LIN {X 0,Y 627.245,Z 767.06,A -85,B 0,C 180,E1 6657.903,E2 6657.903} C_VEL
LIN {X 0,Y 626.761,Z 767.06,A -85,B 0,C 180,E1 6666.234,E2 6666.234} C_VEL
LIN {X 0,Y 626.409,Z 767.06,A -85,B 0,C 180,E1 6674.712,E2 6674.712} C_VEL
LIN {X 0,Y 626.287,Z 767.06,A -85,B 0,C 180,E1 6682.031,E2 6682.031} C_VEL
LIN {X 0,Y 626.18,Z 767.06,A -85,B 0,C 180,E1 6690.73,E2 6690.73} C_VEL
LIN {X 0,Y 626.045,Z 767.06,A -85,B 0,C 180,E1 6698.138,E2 6698.138} C_VEL
LIN {X 0,Y 626.097,Z 767.06,A -85,B 0,C 180,E1 6703.652,E2 6703.652} C_VEL
LIN {X 0,Y 628.32,Z 775.547,A -85,B 0,C 180,E1 6704.191,E2 6704.191} C_VEL
LIN {X 0,Y 630.234,Z 788.438,A -85,B 0,C 180,E1 6704.573,E2 6704.573} C_VEL
LIN {X 0,Y 651.421,Z 829.278,A -85,B 0,C 180,E1 6707.069,E2 6707.069} C_VEL
LIN {X 0,Y 646.587,Z 907.539,A -85,B 0,C 180,E1 6708.986,E2 6708.986} C_VEL
LIN {X 0,Y 639.747,Z 982.775,A -85,B 0,C 180,E1 6712.403,E2 6712.403} C_VEL
LIN {X 0,Y 632.395,Z 1050.27,A -85,B 0,C 180,E1 6717.121,E2 6717.121} C_VEL
LIN {X 0,Y 626.259,Z 1107.378,A -85,B 0,C 180,E1 6722.867,E2 6722.867} C_VEL
LIN {X 0,Y 622.003,Z 1154.489,A -85,B 0,C 180,E1 6729.657,E2 6729.657} C_VEL
LIN {X 0,Y 619.694,Z 1186.305,A -85,B 0,C 180,E1 6736.585,E2 6736.585} C_VEL
LIN {X 0,Y 619.248,Z 1202.946,A -85,B 0,C 180,E1 6742.653,E2 6742.653} C_VEL
LIN {X 0,Y 619.266,Z 1209.424,A -85,B 0,C 180,E1 6747.928,E2 6747.928} C_VEL
LIN {X 0,Y 619.05,Z 1206.761,A -85,B 0,C 180,E1 6754.956,E2 6754.956} C_VEL
LIN {X 0,Y 619.262,Z 1193.655,A -85,B 0,C 180,E1 6761.174,E2 6761.174} C_VEL
LIN {X 0,Y 620.519,Z 1169.572,A -85,B 0,C 180,E1 6767.441,E2 6767.441} C_VEL
LIN {X 0,Y 623.271,Z 1133.468,A -85,B 0,C 180,E1 6773.72,E2 6773.72} C_VEL
LIN {X 0,Y 628.625,Z 1081.833,A -85,B 0,C 180,E1 6779.974,E2 6779.974} C_VEL
LIN {X 0,Y 635.923,Z 1018.771,A -85,B 0,C 180,E1 6785.31,E2 6785.31} C_VEL
LIN {X 0,Y 643.31,Z 949.028,A -85,B 0,C 180,E1 6789.325,E2 6789.325} C_VEL
LIN {X 0,Y 649.136,Z 874.323,A -85,B 0,C 180,E1 6792.011,E2 6792.011} C_VEL
LIN {X 0,Y 650.044,Z 823.777,A -85,B 0,C 180,E1 6793.141,E2 6793.141} C_VEL
LIN {X 0,Y 618.157,Z 767.06,A -85,B 0,C 180,E1 6797.036,E2 6797.036} C_VEL
LIN {X 0,Y 618.384,Z 767.06,A -85,B 0,C 180,E1 6806.522,E2 6806.522} C_VEL
LIN {X 0,Y 618.649,Z 767.06,A -85,B 0,C 180,E1 6814.61,E2 6814.61} C_VEL
LIN {X 0,Y 618.58,Z 767.06,A -85,B 0,C 180,E1 6823.639,E2 6823.639} C_VEL
LIN {X 0,Y 618.828,Z 767.06,A -85,B 0,C 180,E1 6832.27,E2 6832.27} C_VEL
LIN {X 0,Y 618.766,Z 767.06,A -85,B 0,C 180,E1 6840.721,E2 6840.721} C_VEL
LIN {X 0,Y 618.86,Z 767.06,A -85,B 0,C 180,E1 6847.767,E2 6847.767} C_VEL
LIN {X 0,Y 618.363,Z 767.06,A -85,B 0,C 180,E1 6856.406,E2 6856.406} C_VEL
LIN {X 0,Y 618.222,Z 767.06,A -85,B 0,C 180,E1 6865.45,E2 6865.45} C_VEL
LIN {X 0,Y 618.091,Z 767.06,A -85,B 0,C 180,E1 6873.541,E2 6873.541} C_VEL
LIN {X 0,Y 618.177,Z 767.06,A -85,B 0,C 180,E1 6882.465,E2 6882.465} C_VEL
LIN {X 0,Y 618.232,Z 768.464,A -85,B 0,C 180,E1 6890.217,E2 6890.217} C_VEL
LIN {X 0,Y 651.124,Z 828.1,A -85,B 0,C 180,E1 6894.171,E2 6894.171} C_VEL
LIN {X 0,Y 646.571,Z 901.597,A -85,B 0,C 180,E1 6896.097,E2 6896.097} C_VEL
LIN {X 0,Y 639.646,Z 974.672,A -85,B 0,C 180,E1 6899.467,E2 6899.467} C_VEL
LIN {X 0,Y 632.064,Z 1042.701,A -85,B 0,C 180,E1 6904.278,E2 6904.278} C_VEL
LIN {X 0,Y 625.576,Z 1101.407,A -85,B 0,C 180,E1 6910.298,E2 6910.298} C_VEL
LIN {X 0,Y 621.333,Z 1147.196,A -85,B 0,C 180,E1 6917.086,E2 6917.086} C_VEL
LIN {X 0,Y 619.437,Z 1176.669,A -85,B 0,C 180,E1 6923.637,E2 6923.637} C_VEL
LIN {X 0,Y 618.869,Z 1193.621,A -85,B 0,C 180,E1 6929.965,E2 6929.965} C_VEL
LIN {X 0,Y 618.768,Z 1199.851,A -85,B 0,C 180,E1 6936.3,E2 6936.3} C_VEL
LIN {X 0,Y 618.868,Z 1195.665,A -85,B 0,C 180,E1 6942.712,E2 6942.712} C_VEL
LIN {X 0,Y 619.249,Z 1179.816,A -85,B 0,C 180,E1 6949.363,E2 6949.363} C_VEL
LIN {X 0,Y 620.829,Z 1153.329,A -85,B 0,C 180,E1 6955.671,E2 6955.671} C_VEL
LIN {X 0,Y 624.482,Z 1111.503,A -85,B 0,C 180,E1 6962.324,E2 6962.324} C_VEL
LIN {X 0,Y 630.592,Z 1055.076,A -85,B 0,C 180,E1 6968.544,E2 6968.544} C_VEL
LIN {X 0,Y 638.132,Z 989.06,A -85,B 0,C 180,E1 6973.576,E2 6973.576} C_VEL
LIN {X 0,Y 645.271,Z 917.737,A -85,B 0,C 180,E1 6977.198,E2 6977.198} C_VEL
LIN {X 0,Y 650.203,Z 848.201,A -85,B 0,C 180,E1 6979.337,E2 6979.337} C_VEL
LIN {X 0,Y 649.666,Z 822.506,A -85,B 0,C 180,E1 6979.978,E2 6979.978} C_VEL
LIN {X 0,Y 618.29,Z 767.06,A -85,B 0,C 180,E1 6983.94,E2 6983.94} C_VEL
LIN {X 0,Y 618.29,Z 767.06,A -85,B 0,C 180,E1 6992.986,E2 6992.986} C_VEL
LIN {X 0,Y 618.359,Z 767.06,A -85,B 0,C 180,E1 7000.747,E2 7000.747} C_VEL
LIN {X 0,Y 619.19,Z 767.06,A -85,B 0,C 180,E1 7009.393,E2 7009.393} C_VEL
LIN {X 0,Y 619.243,Z 767.06,A -85,B 0,C 180,E1 7017.876,E2 7017.876} C_VEL
LIN {X 0,Y 618.542,Z 767.06,A -85,B 0,C 180,E1 7026.854,E2 7026.854} C_VEL
LIN {X 0,Y 618.36,Z 767.06,A -85,B 0,C 180,E1 7034.908,E2 7034.908} C_VEL
LIN {X 0,Y 618.08,Z 767.06,A -85,B 0,C 180,E1 7043.081,E2 7043.081} C_VEL
LIN {X 0,Y 618.03,Z 767.06,A -85,B 0,C 180,E1 7051.829,E2 7051.829} C_VEL
LIN {X 0,Y 617.761,Z 767.06,A -85,B 0,C 180,E1 7060.572,E2 7060.572} C_VEL
LIN {X 0,Y 618.103,Z 768.608,A -85,B 0,C 180,E1 7063.099,E2 7063.099} C_VEL
LIN {X 0,Y 630.234,Z 788.438,A -85,B 0,C 180,E1 7064.573,E2 7064.573} C_VEL
LIN {X 0,Y 635.159,Z 810.265,A -85,B 0,C 180,E1 7065.359,E2 7065.359} C_VEL
LIN {X 0,Y 645.533,Z 832.217,A -85,B 0,C 180,E1 7066.634,E2 7066.634} C_VEL
LIN {X 0,Y 640.352,Z 909.412,A -85,B 0,C 180,E1 7068.575,E2 7068.575} C_VEL
LIN {X 0,Y 633.189,Z 982.863,A -85,B 0,C 180,E1 7071.95,E2 7071.95} C_VEL
LIN {X 0,Y 625.431,Z 1049.905,A -85,B 0,C 180,E1 7076.674,E2 7076.674} C_VEL
LIN {X 0,Y 618.742,Z 1107.804,A -85,B 0,C 180,E1 7082.563,E2 7082.563} C_VEL
LIN {X 0,Y 614.293,Z 1154.485,A -85,B 0,C 180,E1 7089.389,E2 7089.389} C_VEL
LIN {X 0,Y 611.622,Z 1187.618,A -85,B 0,C 180,E1 7096.77,E2 7096.77} C_VEL
LIN {X 0,Y 610.939,Z 1204.79,A -85,B 0,C 180,E1 7103.619,E2 7103.619} C_VEL
LIN {X 0,Y 610.73,Z 1209.846,A -85,B 0,C 180,E1 7109.323,E2 7109.323} C_VEL
LIN {X 0,Y 610.928,Z 1205.826,A -85,B 0,C 180,E1 7115.737,E2 7115.737} C_VEL
LIN {X 0,Y 611.291,Z 1190.908,A -85,B 0,C 180,E1 7122.215,E2 7122.215} C_VEL
LIN {X 0,Y 612.788,Z 1165.943,A -85,B 0,C 180,E1 7128.439,E2 7128.439} C_VEL
LIN {X 0,Y 616.388,Z 1126.344,A -85,B 0,C 180,E1 7135.04,E2 7135.04} C_VEL
LIN {X 0,Y 622.443,Z 1072.303,A -85,B 0,C 180,E1 7141.31,E2 7141.31} C_VEL
LIN {X 0,Y 630.415,Z 1007.933,A -85,B 0,C 180,E1 7146.495,E2 7146.495} C_VEL
LIN {X 0,Y 638.116,Z 938.064,A -85,B 0,C 180,E1 7150.277,E2 7150.277} C_VEL
LIN {X 0,Y 643.685,Z 867.024,A -85,B 0,C 180,E1 7152.661,E2 7152.661} C_VEL
LIN {X 0,Y 644.21,Z 827.262,A -85,B 0,C 180,E1 7153.566,E2 7153.566} C_VEL
LIN {X 0,Y 610.074,Z 767.06,A -85,B 0,C 180,E1 7157.871,E2 7157.871} C_VEL
LIN {X 0,Y 610.378,Z 767.06,A -85,B 0,C 180,E1 7166.445,E2 7166.445} C_VEL
LIN {X 0,Y 610.572,Z 767.06,A -85,B 0,C 180,E1 7175.181,E2 7175.181} C_VEL
LIN {X 0,Y 610.494,Z 767.06,A -85,B 0,C 180,E1 7184.896,E2 7184.896} C_VEL
LIN {X 0,Y 610.475,Z 767.06,A -85,B 0,C 180,E1 7193.599,E2 7193.599} C_VEL
LIN {X 0,Y 610.759,Z 767.06,A -85,B 0,C 180,E1 7200.73,E2 7200.73} C_VEL
LIN {X 0,Y 610.807,Z 767.06,A -85,B 0,C 180,E1 7207.87,E2 7207.87} C_VEL
LIN {X 0,Y 610.277,Z 767.06,A -85,B 0,C 180,E1 7216.704,E2 7216.704} C_VEL
LIN {X 0,Y 610.235,Z 767.06,A -85,B 0,C 180,E1 7224.751,E2 7224.751} C_VEL
LIN {X 0,Y 610.105,Z 767.06,A -85,B 0,C 180,E1 7233.517,E2 7233.517} C_VEL
LIN {X 0,Y 610.171,Z 767.06,A -85,B 0,C 180,E1 7242.763,E2 7242.763} C_VEL
LIN {X 0,Y 610.117,Z 768.406,A -85,B 0,C 180,E1 7249.401,E2 7249.401} C_VEL
LIN {X 0,Y 645.164,Z 829.949,A -85,B 0,C 180,E1 7253.722,E2 7253.722} C_VEL
LIN {X 0,Y 640.323,Z 902.679,A -85,B 0,C 180,E1 7255.661,E2 7255.661} C_VEL
LIN {X 0,Y 632.989,Z 975.5,A -85,B 0,C 180,E1 7259.06,E2 7259.06} C_VEL
LIN {X 0,Y 625.052,Z 1042.571,A -85,B 0,C 180,E1 7263.853,E2 7263.853} C_VEL
LIN {X 0,Y 618.218,Z 1100.711,A -85,B 0,C 180,E1 7269.867,E2 7269.867} C_VEL
LIN {X 0,Y 613.633,Z 1146.761,A -85,B 0,C 180,E1 7276.743,E2 7276.743} C_VEL
LIN {X 0,Y 611.514,Z 1176.997,A -85,B 0,C 180,E1 7283.554,E2 7283.554} C_VEL
LIN {X 0,Y 610.885,Z 1193.782,A -85,B 0,C 180,E1 7289.965,E2 7289.965} C_VEL
LIN {X 0,Y 610.775,Z 1199.873,A -85,B 0,C 180,E1 7296.383,E2 7296.383} C_VEL
LIN {X 0,Y 610.899,Z 1195.518,A -85,B 0,C 180,E1 7302.88,E2 7302.88} C_VEL
LIN {X 0,Y 611.328,Z 1179.774,A -85,B 0,C 180,E1 7309.539,E2 7309.539} C_VEL
LIN {X 0,Y 613.078,Z 1152.806,A -85,B 0,C 180,E1 7316.019,E2 7316.019} C_VEL
LIN {X 0,Y 617.224,Z 1109.621,A -85,B 0,C 180,E1 7322.904,E2 7322.904} C_VEL
LIN {X 0,Y 623.652,Z 1053.919,A -85,B 0,C 180,E1 7329.053,E2 7329.053} C_VEL
LIN {X 0,Y 631.741,Z 986.989,A -85,B 0,C 180,E1 7334.155,E2 7334.155} C_VEL
LIN {X 0,Y 639.21,Z 915.736,A -85,B 0,C 180,E1 7337.752,E2 7337.752} C_VEL
LIN {X 0,Y 644.327,Z 847.615,A -85,B 0,C 180,E1 7339.831,E2 7339.831} C_VEL
LIN {X 0,Y 643.853,Z 826.122,A -85,B 0,C 180,E1 7340.385,E2 7340.385} C_VEL
LIN {X 0,Y 610.198,Z 767.06,A -85,B 0,C 180,E1 7344.645,E2 7344.645} C_VEL
LIN {X 0,Y 610.258,Z 767.06,A -85,B 0,C 180,E1 7352.601,E2 7352.601} C_VEL
LIN {X 0,Y 610.343,Z 767.06,A -85,B 0,C 180,E1 7360.375,E2 7360.375} C_VEL
LIN {X 0,Y 611.184,Z 767.06,A -85,B 0,C 180,E1 7369.253,E2 7369.253} C_VEL
LIN {X 0,Y 611.254,Z 767.06,A -85,B 0,C 180,E1 7377.848,E2 7377.848} C_VEL
LIN {X 0,Y 610.687,Z 767.06,A -85,B 0,C 180,E1 7386.399,E2 7386.399} C_VEL
LIN {X 0,Y 610.305,Z 767.06,A -85,B 0,C 180,E1 7395.109,E2 7395.109} C_VEL
LIN {X 0,Y 610.146,Z 767.06,A -85,B 0,C 180,E1 7402.646,E2 7402.646} C_VEL
LIN {X 0,Y 610.077,Z 767.06,A -85,B 0,C 180,E1 7410.973,E2 7410.973} C_VEL
LIN {X 0,Y 609.847,Z 767.06,A -85,B 0,C 180,E1 7419.343,E2 7419.343} C_VEL
LIN {X 0,Y 610.08,Z 768.922,A -85,B 0,C 180,E1 7422.298,E2 7422.298} C_VEL
LIN {X 0,Y 635.159,Z 810.265,A -85,B 0,C 180,E1 7425.359,E2 7425.359} C_VEL
LIN {X 0,Y 639.562,Z 835.031,A -85,B 0,C 180,E1 7426.178,E2 7426.178} C_VEL
LIN {X 0,Y 639.2,Z 843.944,A -85,B 0,C 180,E1 7426.355,E2 7426.355} C_VEL
LIN {X 0,Y 633.542,Z 919,A -85,B 0,C 180,E1 7428.451,E2 7428.451} C_VEL
LIN {X 0,Y 625.551,Z 992.775,A -85,B 0,C 180,E1 7432.078,E2 7432.078} C_VEL
LIN {X 0,Y 617.373,Z 1058.589,A -85,B 0,C 180,E1 7437.016,E2 7437.016} C_VEL
LIN {X 0,Y 610.525,Z 1114.591,A -85,B 0,C 180,E1 7443.061,E2 7443.061} C_VEL
LIN {X 0,Y 605.801,Z 1159.36,A -85,B 0,C 180,E1 7450.023,E2 7450.023} C_VEL
LIN {X 0,Y 603.549,Z 1188.827,A -85,B 0,C 180,E1 7456.96,E2 7456.96} C_VEL
LIN {X 0,Y 602.979,Z 1204.787,A -85,B 0,C 180,E1 7463.534,E2 7463.534} C_VEL
LIN {X 0,Y 602.732,Z 1209.846,A -85,B 0,C 180,E1 7469.314,E2 7469.314} C_VEL
LIN {X 0,Y 602.939,Z 1205.826,A -85,B 0,C 180,E1 7475.813,E2 7475.813} C_VEL
LIN {X 0,Y 603.328,Z 1190.905,A -85,B 0,C 180,E1 7482.379,E2 7482.379} C_VEL
LIN {X 0,Y 604.93,Z 1165.944,A -85,B 0,C 180,E1 7488.688,E2 7488.688} C_VEL
LIN {X 0,Y 608.833,Z 1125.749,A -85,B 0,C 180,E1 7495.46,E2 7495.46} C_VEL
LIN {X 0,Y 615.417,Z 1071.635,A -85,B 0,C 180,E1 7501.781,E2 7501.781} C_VEL
LIN {X 0,Y 623.853,Z 1007.033,A -85,B 0,C 180,E1 7507.013,E2 7507.013} C_VEL
LIN {X 0,Y 631.918,Z 937.652,A -85,B 0,C 180,E1 7510.776,E2 7510.776} C_VEL
LIN {X 0,Y 637.734,Z 867.851,A -85,B 0,C 180,E1 7513.131,E2 7513.131} C_VEL
LIN {X 0,Y 638.364,Z 830.573,A -85,B 0,C 180,E1 7514.006,E2 7514.006} C_VEL
LIN {X 0,Y 602.051,Z 767.06,A -85,B 0,C 180,E1 7518.785,E2 7518.785} C_VEL
LIN {X 0,Y 602.457,Z 767.06,A -85,B 0,C 180,E1 7527.598,E2 7527.598} C_VEL
LIN {X 0,Y 602.587,Z 767.06,A -85,B 0,C 180,E1 7535.478,E2 7535.478} C_VEL
LIN {X 0,Y 602.487,Z 767.06,A -85,B 0,C 180,E1 7544.69,E2 7544.69} C_VEL
LIN {X 0,Y 602.485,Z 767.06,A -85,B 0,C 180,E1 7553.513,E2 7553.513} C_VEL
LIN {X 0,Y 602.751,Z 767.06,A -85,B 0,C 180,E1 7560.74,E2 7560.74} C_VEL
LIN {X 0,Y 602.77,Z 767.06,A -85,B 0,C 180,E1 7567.975,E2 7567.975} C_VEL
LIN {X 0,Y 602.259,Z 767.06,A -85,B 0,C 180,E1 7576.857,E2 7576.857} C_VEL
LIN {X 0,Y 602.251,Z 767.06,A -85,B 0,C 180,E1 7584.578,E2 7584.578} C_VEL
LIN {X 0,Y 602.113,Z 767.06,A -85,B 0,C 180,E1 7592.82,E2 7592.82} C_VEL
LIN {X 0,Y 602.098,Z 767.06,A -85,B 0,C 180,E1 7601.926,E2 7601.926} C_VEL
LIN {X 0,Y 602.207,Z 768.812,A -85,B 0,C 180,E1 7608.58,E2 7608.58} C_VEL
LIN {X 0,Y 639.091,Z 832.378,A -85,B 0,C 180,E1 7613.264,E2 7613.264} C_VEL
LIN {X 0,Y 633.97,Z 905.735,A -85,B 0,C 180,E1 7615.294,E2 7615.294} C_VEL
LIN {X 0,Y 626.169,Z 978.142,A -85,B 0,C 180,E1 7618.756,E2 7618.756} C_VEL
LIN {X 0,Y 617.745,Z 1044.932,A -85,B 0,C 180,E1 7623.637,E2 7623.637} C_VEL
LIN {X 0,Y 610.474,Z 1102.98,A -85,B 0,C 180,E1 7629.79,E2 7629.79} C_VEL
LIN {X 0,Y 605.819,Z 1147.273,A -85,B 0,C 180,E1 7636.568,E2 7636.568} C_VEL
LIN {X 0,Y 603.594,Z 1177.326,A -85,B 0,C 180,E1 7643.469,E2 7643.469} C_VEL
LIN {X 0,Y 602.884,Z 1193.93,A -85,B 0,C 180,E1 7649.964,E2 7649.964} C_VEL
LIN {X 0,Y 602.78,Z 1199.894,A -85,B 0,C 180,E1 7656.468,E2 7656.468} C_VEL
LIN {X 0,Y 602.918,Z 1195.37,A -85,B 0,C 180,E1 7663.054,E2 7663.054} C_VEL
LIN {X 0,Y 603.442,Z 1179.466,A -85,B 0,C 180,E1 7669.805,E2 7669.805} C_VEL
LIN {X 0,Y 605.789,Z 1149.32,A -85,B 0,C 180,E1 7676.949,E2 7676.949} C_VEL
LIN {X 0,Y 610.52,Z 1104.186,A -85,B 0,C 180,E1 7683.956,E2 7683.956} C_VEL
LIN {X 0,Y 617.47,Z 1047.599,A -85,B 0,C 180,E1 7690.034,E2 7690.034} C_VEL
LIN {X 0,Y 625.867,Z 980.636,A -85,B 0,C 180,E1 7695.003,E2 7695.003} C_VEL
LIN {X 0,Y 633.785,Z 907.439,A -85,B 0,C 180,E1 7698.553,E2 7698.553} C_VEL
LIN {X 0,Y 639.125,Z 835.51,A -85,B 0,C 180,E1 7700.571,E2 7700.571} C_VEL
LIN {X 0,Y 612.906,Z 785.364,A -85,B 0,C 180,E1 7703.938,E2 7703.938} C_VEL
LIN {X 0,Y 602.132,Z 767.06,A -85,B 0,C 180,E1 7705.447,E2 7705.447} C_VEL
LIN {X 0,Y 602.207,Z 767.06,A -85,B 0,C 180,E1 7713.823,E2 7713.823} C_VEL
LIN {X 0,Y 602.301,Z 767.06,A -85,B 0,C 180,E1 7721.63,E2 7721.63} C_VEL
LIN {X 0,Y 603.206,Z 767.06,A -85,B 0,C 180,E1 7729.109,E2 7729.109} C_VEL
LIN {X 0,Y 603.25,Z 767.06,A -85,B 0,C 180,E1 7737.819,E2 7737.819} C_VEL
LIN {X 0,Y 602.65,Z 767.06,A -85,B 0,C 180,E1 7746.485,E2 7746.485} C_VEL
LIN {X 0,Y 602.256,Z 767.06,A -85,B 0,C 180,E1 7755.316,E2 7755.316} C_VEL
LIN {X 0,Y 602.056,Z 767.06,A -85,B 0,C 180,E1 7763.186,E2 7763.186} C_VEL
LIN {X 0,Y 602.073,Z 767.06,A -85,B 0,C 180,E1 7771.076,E2 7771.076} C_VEL
LIN {X 0,Y 601.779,Z 767.06,A -85,B 0,C 180,E1 7779.976,E2 7779.976} C_VEL
LIN {X 0,Y 601.935,Z 768.669,A -85,B 0,C 180,E1 7781.426,E2 7781.426} C_VEL
LIN {X 0,Y 639.583,Z 833.093,A -85,B 0,C 180,E1 7786.145,E2 7786.145} C_VEL
LIN {X 0,Y 639.2,Z 843.944,A -85,B 0,C 180,E1 7786.355,E2 7786.355} C_VEL
LIN {X 0,Y 631.176,Z 878.377,A -85,B 0,C 180,E1 7786.642,E2 7786.642} C_VEL
LIN {X 0,Y 624.414,Z 949.498,A -85,B 0,C 180,E1 7789.265,E2 7789.265} C_VEL
LIN {X 0,Y 615.761,Z 1018.278,A -85,B 0,C 180,E1 7793.312,E2 7793.312} C_VEL
LIN {X 0,Y 606.941,Z 1082.187,A -85,B 0,C 180,E1 7798.877,E2 7798.877} C_VEL
LIN {X 0,Y 600.372,Z 1133.976,A -85,B 0,C 180,E1 7805.394,E2 7805.394} C_VEL
LIN {X 0,Y 596.774,Z 1170.294,A -85,B 0,C 180,E1 7812,E2 7812} C_VEL
LIN {X 0,Y 595.208,Z 1193.25,A -85,B 0,C 180,E1 7818.224,E2 7818.224} C_VEL
LIN {X 0,Y 594.961,Z 1206.836,A -85,B 0,C 180,E1 7824.915,E2 7824.915} C_VEL
LIN {X 0,Y 594.613,Z 1209.829,A -85,B 0,C 180,E1 7830.767,E2 7830.767} C_VEL
LIN {X 0,Y 594.994,Z 1204.665,A -85,B 0,C 180,E1 7836.626,E2 7836.626} C_VEL
LIN {X 0,Y 595.769,Z 1187.377,A -85,B 0,C 180,E1 7843.662,E2 7843.662} C_VEL
LIN {X 0,Y 598.604,Z 1155.322,A -85,B 0,C 180,E1 7851.019,E2 7851.019} C_VEL
LIN {X 0,Y 603.669,Z 1109.45,A -85,B 0,C 180,E1 7857.973,E2 7857.973} C_VEL
LIN {X 0,Y 611.225,Z 1052.148,A -85,B 0,C 180,E1 7863.996,E2 7863.996} C_VEL
LIN {X 0,Y 620.033,Z 985.616,A -85,B 0,C 180,E1 7868.826,E2 7868.826} C_VEL
LIN {X 0,Y 628.218,Z 911.551,A -85,B 0,C 180,E1 7872.319,E2 7872.319} C_VEL
LIN {X 0,Y 632.404,Z 833.705,A -85,B 0,C 180,E1 7874.47,E2 7874.47} C_VEL
LIN {X 0,Y 596.309,Z 772.647,A -85,B 0,C 180,E1 7879.091,E2 7879.091} C_VEL
LIN {X 0,Y 594.044,Z 767.06,A -85,B 0,C 180,E1 7879.633,E2 7879.633} C_VEL
LIN {X 0,Y 594.49,Z 767.06,A -85,B 0,C 180,E1 7888.829,E2 7888.829} C_VEL
LIN {X 0,Y 594.409,Z 767.06,A -85,B 0,C 180,E1 7896.72,E2 7896.72} C_VEL
LIN {X 0,Y 594.331,Z 767.06,A -85,B 0,C 180,E1 7905.987,E2 7905.987} C_VEL
LIN {X 0,Y 594.496,Z 767.06,A -85,B 0,C 180,E1 7913.426,E2 7913.426} C_VEL
LIN {X 0,Y 594.751,Z 767.06,A -85,B 0,C 180,E1 7920.75,E2 7920.75} C_VEL
LIN {X 0,Y 594.722,Z 767.06,A -85,B 0,C 180,E1 7928.084,E2 7928.084} C_VEL
LIN {X 0,Y 594.233,Z 767.06,A -85,B 0,C 180,E1 7937.092,E2 7937.092} C_VEL
LIN {X 0,Y 594.206,Z 767.06,A -85,B 0,C 180,E1 7944.933,E2 7944.933} C_VEL
LIN {X 0,Y 594.014,Z 767.06,A -85,B 0,C 180,E1 7953.822,E2 7953.822} C_VEL
LIN {X 0,Y 594.061,Z 767.06,A -85,B 0,C 180,E1 7962.611,E2 7962.611} C_VEL
LIN {X 0,Y 594.184,Z 768.882,A -85,B 0,C 180,E1 7967.721,E2 7967.721} C_VEL
LIN {X 0,Y 632.996,Z 835.271,A -85,B 0,C 180,E1 7972.803,E2 7972.803} C_VEL
LIN {X 0,Y 627.613,Z 908.776,A -85,B 0,C 180,E1 7974.917,E2 7974.917} C_VEL
LIN {X 0,Y 619.346,Z 981.073,A -85,B 0,C 180,E1 7978.465,E2 7978.465} C_VEL
LIN {X 0,Y 610.427,Z 1047.351,A -85,B 0,C 180,E1 7983.42,E2 7983.42} C_VEL
LIN {X 0,Y 602.938,Z 1103.755,A -85,B 0,C 180,E1 7989.526,E2 7989.526} C_VEL
LIN {X 0,Y 598.024,Z 1147.784,A -85,B 0,C 180,E1 7996.39,E2 7996.39} C_VEL
LIN {X 0,Y 595.649,Z 1177.655,A -85,B 0,C 180,E1 8003.382,E2 8003.382} C_VEL
LIN {X 0,Y 594.889,Z 1194.078,A -85,B 0,C 180,E1 8009.964,E2 8009.964} C_VEL
LIN {X 0,Y 594.772,Z 1199.916,A -85,B 0,C 180,E1 8016.556,E2 8016.556} C_VEL
LIN {X 0,Y 594.972,Z 1195.22,A -85,B 0,C 180,E1 8023.231,E2 8023.231} C_VEL
LIN {X 0,Y 595.828,Z 1177.885,A -85,B 0,C 180,E1 8030.458,E2 8030.458} C_VEL
LIN {X 0,Y 598.642,Z 1145.555,A -85,B 0,C 180,E1 8037.922,E2 8037.922} C_VEL
LIN {X 0,Y 603.781,Z 1098.812,A -85,B 0,C 180,E1 8044.996,E2 8044.996} C_VEL
LIN {X 0,Y 611.28,Z 1042.076,A -85,B 0,C 180,E1 8050.95,E2 8050.95} C_VEL
LIN {X 0,Y 620.132,Z 974.657,A -85,B 0,C 180,E1 8055.839,E2 8055.839} C_VEL
LIN {X 0,Y 628.372,Z 899.804,A -85,B 0,C 180,E1 8059.344,E2 8059.344} C_VEL
LIN {X 0,Y 632.022,Z 833.034,A -85,B 0,C 180,E1 8061.246,E2 8061.246} C_VEL
LIN {X 0,Y 595.921,Z 772.134,A -85,B 0,C 180,E1 8065.99,E2 8065.99} C_VEL
LIN {X 0,Y 594.118,Z 767.06,A -85,B 0,C 180,E1 8066.387,E2 8066.387} C_VEL
LIN {X 0,Y 594.254,Z 767.06,A -85,B 0,C 180,E1 8075.069,E2 8075.069} C_VEL
LIN {X 0,Y 594.762,Z 767.06,A -85,B 0,C 180,E1 8084.446,E2 8084.446} C_VEL
LIN {X 0,Y 594.508,Z 767.06,A -85,B 0,C 180,E1 8091.913,E2 8091.913} C_VEL
LIN {X 0,Y 594.626,Z 767.06,A -85,B 0,C 180,E1 8099.25,E2 8099.25} C_VEL
LIN {X 0,Y 594.614,Z 767.06,A -85,B 0,C 180,E1 8106.573,E2 8106.573} C_VEL
LIN {X 0,Y 594.219,Z 767.06,A -85,B 0,C 180,E1 8115.528,E2 8115.528} C_VEL
LIN {X 0,Y 594.036,Z 767.06,A -85,B 0,C 180,E1 8123.296,E2 8123.296} C_VEL
LIN {X 0,Y 594.015,Z 767.06,A -85,B 0,C 180,E1 8131.546,E2 8131.546} C_VEL
LIN {X 0,Y 593.804,Z 767.957,A -85,B 0,C 180,E1 8140.485,E2 8140.485} C_VEL
LIN {X 0,Y 632.52,Z 834.054,A -85,B 0,C 180,E1 8145.547,E2 8145.547} C_VEL
LIN {X 0,Y 631.176,Z 878.377,A -85,B 0,C 180,E1 8146.642,E2 8146.642} C_VEL
LIN {X 0,Y 621.987,Z 912.08,A -85,B 0,C 180,E1 8147.179,E2 8147.179} C_VEL
LIN {X 0,Y 613.377,Z 987.22,A -85,B 0,C 180,E1 8150.781,E2 8150.781} C_VEL
LIN {X 0,Y 604.04,Z 1054.15,A -85,B 0,C 180,E1 8155.735,E2 8155.735} C_VEL
LIN {X 0,Y 595.986,Z 1111.693,A -85,B 0,C 180,E1 8161.943,E2 8161.943} C_VEL
LIN {X 0,Y 590.824,Z 1156.722,A -85,B 0,C 180,E1 8168.968,E2 8168.968} C_VEL
LIN {X 0,Y 587.761,Z 1188.825,A -85,B 0,C 180,E1 8176.603,E2 8176.603} C_VEL
LIN {X 0,Y 587.056,Z 1204.781,A -85,B 0,C 180,E1 8183.358,E2 8183.358} C_VEL
LIN {X 0,Y 586.736,Z 1209.846,A -85,B 0,C 180,E1 8189.296,E2 8189.296} C_VEL
LIN {X 0,Y 586.959,Z 1205.894,A -85,B 0,C 180,E1 8195.923,E2 8195.923} C_VEL
LIN {X 0,Y 587.452,Z 1190.899,A -85,B 0,C 180,E1 8202.719,E2 8202.719} C_VEL
LIN {X 0,Y 589.512,Z 1164.357,A -85,B 0,C 180,E1 8209.546,E2 8209.546} C_VEL
LIN {X 0,Y 594.461,Z 1121.344,A -85,B 0,C 180,E1 8216.778,E2 8216.778} C_VEL
LIN {X 0,Y 602.182,Z 1066.118,A -85,B 0,C 180,E1 8223.153,E2 8223.153} C_VEL
LIN {X 0,Y 611.544,Z 1000.886,A -85,B 0,C 180,E1 8228.352,E2 8228.352} C_VEL
LIN {X 0,Y 620.473,Z 929.697,A -85,B 0,C 180,E1 8232.107,E2 8232.107} C_VEL
LIN {X 0,Y 626.537,Z 861.693,A -85,B 0,C 180,E1 8234.281,E2 8234.281} C_VEL
LIN {X 0,Y 626.492,Z 836.828,A -85,B 0,C 180,E1 8234.934,E2 8234.934} C_VEL
LIN {X 0,Y 591.213,Z 777.282,A -85,B 0,C 180,E1 8239.56,E2 8239.56} C_VEL
LIN {X 0,Y 586.089,Z 767.06,A -85,B 0,C 180,E1 8240.479,E2 8240.479} C_VEL
LIN {X 0,Y 586.464,Z 767.06,A -85,B 0,C 180,E1 8249.732,E2 8249.732} C_VEL
LIN {X 0,Y 586.185,Z 767.06,A -85,B 0,C 180,E1 8257.982,E2 8257.982} C_VEL
LIN {X 0,Y 586.323,Z 767.06,A -85,B 0,C 180,E1 8266.18,E2 8266.18} C_VEL
LIN {X 0,Y 586.528,Z 767.06,A -85,B 0,C 180,E1 8273.336,E2 8273.336} C_VEL
LIN {X 0,Y 586.744,Z 767.06,A -85,B 0,C 180,E1 8280.76,E2 8280.76} C_VEL
LIN {X 0,Y 586.674,Z 767.06,A -85,B 0,C 180,E1 8288.196,E2 8288.196} C_VEL
LIN {X 0,Y 586.18,Z 767.06,A -85,B 0,C 180,E1 8297.334,E2 8297.334} C_VEL
LIN {X 0,Y 586.159,Z 767.06,A -85,B 0,C 180,E1 8305.3,E2 8305.3} C_VEL
LIN {X 0,Y 586.013,Z 767.06,A -85,B 0,C 180,E1 8313.841,E2 8313.841} C_VEL
LIN {X 0,Y 586.083,Z 767.06,A -85,B 0,C 180,E1 8323.333,E2 8323.333} C_VEL
LIN {X 0,Y 586.053,Z 768.171,A -85,B 0,C 180,E1 8326.812,E2 8326.812} C_VEL
LIN {X 0,Y 626.457,Z 837.296,A -85,B 0,C 180,E1 8332.267,E2 8332.267} C_VEL
LIN {X 0,Y 621.185,Z 912.919,A -85,B 0,C 180,E1 8334.576,E2 8334.576} C_VEL
LIN {X 0,Y 612.385,Z 984.847,A -85,B 0,C 180,E1 8338.215,E2 8338.215} C_VEL
LIN {X 0,Y 602.979,Z 1050.931,A -85,B 0,C 180,E1 8343.307,E2 8343.307} C_VEL
LIN {X 0,Y 594.995,Z 1107.354,A -85,B 0,C 180,E1 8349.63,E2 8349.63} C_VEL
LIN {X 0,Y 589.921,Z 1150.222,A -85,B 0,C 180,E1 8356.578,E2 8356.578} C_VEL
LIN {X 0,Y 587.507,Z 1179.592,A -85,B 0,C 180,E1 8363.792,E2 8363.792} C_VEL
LIN {X 0,Y 586.893,Z 1194.226,A -85,B 0,C 180,E1 8369.963,E2 8369.963} C_VEL
LIN {X 0,Y 586.783,Z 1199.937,A -85,B 0,C 180,E1 8376.645,E2 8376.645} C_VEL
LIN {X 0,Y 587.013,Z 1195.064,A -85,B 0,C 180,E1 8383.414,E2 8383.414} C_VEL
LIN {X 0,Y 587.996,Z 1177.535,A -85,B 0,C 180,E1 8390.743,E2 8390.743} C_VEL
LIN {X 0,Y 590.898,Z 1144.962,A -85,B 0,C 180,E1 8398.32,E2 8398.32} C_VEL
LIN {X 0,Y 596.509,Z 1097.699,A -85,B 0,C 180,E1 8405.517,E2 8405.517} C_VEL
LIN {X 0,Y 604.705,Z 1039.478,A -85,B 0,C 180,E1 8411.628,E2 8411.628} C_VEL
LIN {X 0,Y 614.104,Z 971.714,A -85,B 0,C 180,E1 8416.501,E2 8416.501} C_VEL
LIN {X 0,Y 622.573,Z 896.871,A -85,B 0,C 180,E1 8419.955,E2 8419.955} C_VEL
LIN {X 0,Y 625.977,Z 836.196,A -85,B 0,C 180,E1 8421.713,E2 8421.713} C_VEL
LIN {X 0,Y 589.109,Z 773.305,A -85,B 0,C 180,E1 8426.774,E2 8426.774} C_VEL
LIN {X 0,Y 586.099,Z 767.06,A -85,B 0,C 180,E1 8427.271,E2 8427.271} C_VEL
LIN {X 0,Y 586.401,Z 767.06,A -85,B 0,C 180,E1 8436.621,E2 8436.621} C_VEL
LIN {X 0,Y 586.98,Z 767.06,A -85,B 0,C 180,E1 8445.768,E2 8445.768} C_VEL
LIN {X 0,Y 586.464,Z 767.06,A -85,B 0,C 180,E1 8454.511,E2 8454.511} C_VEL
LIN {X 0,Y 586.374,Z 767.06,A -85,B 0,C 180,E1 8460.722,E2 8460.722} C_VEL
LIN {X 0,Y 586.299,Z 767.06,A -85,B 0,C 180,E1 8468.161,E2 8468.161} C_VEL
LIN {X 0,Y 586.194,Z 767.06,A -85,B 0,C 180,E1 8475.746,E2 8475.746} C_VEL
LIN {X 0,Y 586.004,Z 767.06,A -85,B 0,C 180,E1 8483.634,E2 8483.634} C_VEL
LIN {X 0,Y 585.933,Z 767.06,A -85,B 0,C 180,E1 8492.032,E2 8492.032} C_VEL
LIN {X 0,Y 585.964,Z 768.676,A -85,B 0,C 180,E1 8499.547,E2 8499.547} C_VEL
LIN {X 0,Y 623.451,Z 830.848,A -85,B 0,C 180,E1 8504.669,E2 8504.669} C_VEL
LIN {X 0,Y 627.617,Z 844.209,A -85,B 0,C 180,E1 8505.35,E2 8505.35} C_VEL
LIN {X 0,Y 621.987,Z 912.08,A -85,B 0,C 180,E1 8507.179,E2 8507.179} C_VEL
LIN {X 0,Y 612.643,Z 945.005,A -85,B 0,C 180,E1 8508.062,E2 8508.062} C_VEL
LIN {X 0,Y 603.074,Z 1014.337,A -85,B 0,C 180,E1 8512.086,E2 8512.086} C_VEL
LIN {X 0,Y 593.138,Z 1078.702,A -85,B 0,C 180,E1 8517.676,E2 8517.676} C_VEL
LIN {X 0,Y 585.609,Z 1131.325,A -85,B 0,C 180,E1 8524.32,E2 8524.32} C_VEL
LIN {X 0,Y 581.298,Z 1168.055,A -85,B 0,C 180,E1 8530.997,E2 8530.997} C_VEL
LIN {X 0,Y 579.316,Z 1193.385,A -85,B 0,C 180,E1 8537.943,E2 8537.943} C_VEL
LIN {X 0,Y 578.956,Z 1206.831,A -85,B 0,C 180,E1 8544.774,E2 8544.774} C_VEL
LIN {X 0,Y 578.637,Z 1209.829,A -85,B 0,C 180,E1 8550.788,E2 8550.788} C_VEL
LIN {X 0,Y 579.212,Z 1203.447,A -85,B 0,C 180,E1 8557.563,E2 8557.563} C_VEL
LIN {X 0,Y 580.575,Z 1183.595,A -85,B 0,C 180,E1 8565.119,E2 8565.119} C_VEL
LIN {X 0,Y 583.688,Z 1148.389,A -85,B 0,C 180,E1 8572.871,E2 8572.871} C_VEL
LIN {X 0,Y 590.02,Z 1100.352,A -85,B 0,C 180,E1 8579.876,E2 8579.876} C_VEL
LIN {X 0,Y 599.259,Z 1040.26,A -85,B 0,C 180,E1 8585.917,E2 8585.917} C_VEL
LIN {X 0,Y 609.16,Z 971.654,A -85,B 0,C 180,E1 8590.607,E2 8590.607} C_VEL
LIN {X 0,Y 617.623,Z 895.505,A -85,B 0,C 180,E1 8593.907,E2 8593.907} C_VEL
LIN {X 0,Y 620.589,Z 840.114,A -85,B 0,C 180,E1 8595.393,E2 8595.393} C_VEL
LIN {X 0,Y 584.593,Z 779.001,A -85,B 0,C 180,E1 8600.261,E2 8600.261} C_VEL
LIN {X 0,Y 578.036,Z 767.06,A -85,B 0,C 180,E1 8601.403,E2 8601.403} C_VEL
LIN {X 0,Y 578.383,Z 767.06,A -85,B 0,C 180,E1 8609.264,E2 8609.264} C_VEL
LIN {X 0,Y 578.223,Z 767.06,A -85,B 0,C 180,E1 8617.663,E2 8617.663} C_VEL
LIN {X 0,Y 578.329,Z 767.06,A -85,B 0,C 180,E1 8625.591,E2 8625.591} C_VEL
LIN {X 0,Y 578.534,Z 767.06,A -85,B 0,C 180,E1 8633.244,E2 8633.244} C_VEL
LIN {X 0,Y 578.736,Z 767.06,A -85,B 0,C 180,E1 8640.771,E2 8640.771} C_VEL
LIN {X 0,Y 578.63,Z 767.06,A -85,B 0,C 180,E1 8648.31,E2 8648.31} C_VEL
LIN {X 0,Y 578.133,Z 767.06,A -85,B 0,C 180,E1 8657.583,E2 8657.583} C_VEL
LIN {X 0,Y 578.142,Z 767.06,A -85,B 0,C 180,E1 8665.676,E2 8665.676} C_VEL
LIN {X 0,Y 578.006,Z 767.06,A -85,B 0,C 180,E1 8674.375,E2 8674.375} C_VEL
LIN {X 0,Y 578.072,Z 767.06,A -85,B 0,C 180,E1 8683.744,E2 8683.744} C_VEL
LIN {X 0,Y 578.106,Z 768.386,A -85,B 0,C 180,E1 8685.909,E2 8685.909} C_VEL
LIN {X 0,Y 619.379,Z 838.003,A -85,B 0,C 180,E1 8691.633,E2 8691.633} C_VEL
LIN {X 0,Y 620.846,Z 850.761,A -85,B 0,C 180,E1 8692.125,E2 8692.125} C_VEL
LIN {X 0,Y 614.402,Z 920.581,A -85,B 0,C 180,E1 8694.374,E2 8694.374} C_VEL
LIN {X 0,Y 605.002,Z 991.81,A -85,B 0,C 180,E1 8698.179,E2 8698.179} C_VEL
LIN {X 0,Y 594.962,Z 1057.093,A -85,B 0,C 180,E1 8703.454,E2 8703.454} C_VEL
LIN {X 0,Y 586.75,Z 1112.143,A -85,B 0,C 180,E1 8709.924,E2 8709.924} C_VEL
LIN {X 0,Y 581.828,Z 1152.545,A -85,B 0,C 180,E1 8716.772,E2 8716.772} C_VEL
LIN {X 0,Y 579.506,Z 1180.39,A -85,B 0,C 180,E1 8723.883,E2 8723.883} C_VEL
LIN {X 0,Y 578.907,Z 1194.373,A -85,B 0,C 180,E1 8729.963,E2 8729.963} C_VEL
LIN {X 0,Y 578.775,Z 1199.959,A -85,B 0,C 180,E1 8736.738,E2 8736.738} C_VEL
LIN {X 0,Y 579.042,Z 1194.92,A -85,B 0,C 180,E1 8743.594,E2 8743.594} C_VEL
LIN {X 0,Y 580.304,Z 1176.378,A -85,B 0,C 180,E1 8751.272,E2 8751.272} C_VEL
LIN {X 0,Y 583.306,Z 1142.637,A -85,B 0,C 180,E1 8759.055,E2 8759.055} C_VEL
LIN {X 0,Y 589.36,Z 1095.615,A -85,B 0,C 180,E1 8766.181,E2 8766.181} C_VEL
LIN {X 0,Y 598.347,Z 1036.551,A -85,B 0,C 180,E1 8772.339,E2 8772.339} C_VEL
LIN {X 0,Y 608.054,Z 969.394,A -85,B 0,C 180,E1 8777.129,E2 8777.129} C_VEL
LIN {X 0,Y 616.837,Z 894.746,A -85,B 0,C 180,E1 8780.546,E2 8780.546} C_VEL
LIN {X 0,Y 620.403,Z 840.085,A -85,B 0,C 180,E1 8782.129,E2 8782.129} C_VEL
LIN {X 0,Y 585.318,Z 779.611,A -85,B 0,C 180,E1 8787.118,E2 8787.118} C_VEL
LIN {X 0,Y 578.147,Z 767.06,A -85,B 0,C 180,E1 8788.46,E2 8788.46} C_VEL
LIN {X 0,Y 578.375,Z 767.06,A -85,B 0,C 180,E1 8797.626,E2 8797.626} C_VEL
LIN {X 0,Y 579.131,Z 767.06,A -85,B 0,C 180,E1 8807.115,E2 8807.115} C_VEL
LIN {X 0,Y 579.239,Z 767.06,A -85,B 0,C 180,E1 8817.729,E2 8817.729} C_VEL
LIN {X 0,Y 578.548,Z 767.06,A -85,B 0,C 180,E1 8826.756,E2 8826.756} C_VEL
LIN {X 0,Y 578.405,Z 767.06,A -85,B 0,C 180,E1 8834.407,E2 8834.407} C_VEL
LIN {X 0,Y 578.14,Z 767.06,A -85,B 0,C 180,E1 8842.341,E2 8842.341} C_VEL
LIN {X 0,Y 577.948,Z 767.06,A -85,B 0,C 180,E1 8851.508,E2 8851.508} C_VEL
LIN {X 0,Y 578.006,Z 769.014,A -85,B 0,C 180,E1 8858.529,E2 8858.529} C_VEL
LIN {X 0,Y 615.559,Z 830.048,A -85,B 0,C 180,E1 8863.911,E2 8863.911} C_VEL
LIN {X 0,Y 621.839,Z 845.349,A -85,B 0,C 180,E1 8864.855,E2 8864.855} C_VEL
LIN {X 0,Y 615.145,Z 921.252,A -85,B 0,C 180,E1 8867.032,E2 8867.032} C_VEL
LIN {X 0,Y 612.643,Z 945.005,A -85,B 0,C 180,E1 8868.062,E2 8868.062} C_VEL
LIN {X 0,Y 602.207,Z 976.798,A -85,B 0,C 180,E1 8869.185,E2 8869.185} C_VEL
LIN {X 0,Y 591.882,Z 1043.97,A -85,B 0,C 180,E1 8873.93,E2 8873.93} C_VEL
LIN {X 0,Y 582.243,Z 1103.404,A -85,B 0,C 180,E1 8880.094,E2 8880.094} C_VEL
LIN {X 0,Y 575.743,Z 1150.859,A -85,B 0,C 180,E1 8887.261,E2 8887.261} C_VEL
LIN {X 0,Y 572.561,Z 1185.314,A -85,B 0,C 180,E1 8895.169,E2 8895.169} C_VEL
LIN {X 0,Y 571.352,Z 1203.563,A -85,B 0,C 180,E1 8902.408,E2 8902.408} C_VEL
LIN {X 0,Y 570.753,Z 1209.846,A -85,B 0,C 180,E1 8909.276,E2 8909.276} C_VEL
LIN {X 0,Y 570.975,Z 1205.826,A -85,B 0,C 180,E1 8916.139,E2 8916.139} C_VEL
LIN {X 0,Y 571.593,Z 1190.893,A -85,B 0,C 180,E1 8923.078,E2 8923.078} C_VEL
LIN {X 0,Y 574.22,Z 1163.006,A -85,B 0,C 180,E1 8930.368,E2 8930.368} C_VEL
LIN {X 0,Y 579.915,Z 1119.903,A -85,B 0,C 180,E1 8937.713,E2 8937.713} C_VEL
LIN {X 0,Y 588.633,Z 1063.836,A -85,B 0,C 180,E1 8944.26,E2 8944.26} C_VEL
LIN {X 0,Y 598.94,Z 999.041,A -85,B 0,C 180,E1 8949.453,E2 8949.453} C_VEL
LIN {X 0,Y 608.681,Z 927.157,A -85,B 0,C 180,E1 8953.235,E2 8953.235} C_VEL
LIN {X 0,Y 615.424,Z 857.272,A -85,B 0,C 180,E1 8955.43,E2 8955.43} C_VEL
LIN {X 0,Y 614.356,Z 842.517,A -85,B 0,C 180,E1 8955.919,E2 8955.919} C_VEL
LIN {X 0,Y 577.36,Z 779.754,A -85,B 0,C 180,E1 8961.071,E2 8961.071} C_VEL
LIN {X 0,Y 570.071,Z 767.06,A -85,B 0,C 180,E1 8962.246,E2 8962.246} C_VEL
LIN {X 0,Y 570.385,Z 767.06,A -85,B 0,C 180,E1 8970.55,E2 8970.55} C_VEL
LIN {X 0,Y 570.081,Z 767.06,A -85,B 0,C 180,E1 8978.969,E2 8978.969} C_VEL
LIN {X 0,Y 570.214,Z 767.06,A -85,B 0,C 180,E1 8986.951,E2 8986.951} C_VEL
LIN {X 0,Y 570.331,Z 767.06,A -85,B 0,C 180,E1 8994.679,E2 8994.679} C_VEL
LIN {X 0,Y 570.729,Z 767.06,A -85,B 0,C 180,E1 9000.781,E2 9000.781} C_VEL
LIN {X 0,Y 570.587,Z 767.06,A -85,B 0,C 180,E1 9008.428,E2 9008.428} C_VEL
LIN {X 0,Y 570.328,Z 767.06,A -85,B 0,C 180,E1 9016.238,E2 9016.238} C_VEL
LIN {X 0,Y 570.165,Z 767.06,A -85,B 0,C 180,E1 9024.377,E2 9024.377} C_VEL
LIN {X 0,Y 570.005,Z 767.06,A -85,B 0,C 180,E1 9033.087,E2 9033.087} C_VEL
LIN {X 0,Y 569.978,Z 767.06,A -85,B 0,C 180,E1 9040.723,E2 9040.723} C_VEL
LIN {X 0,Y 570.044,Z 768.042,A -85,B 0,C 180,E1 9044.947,E2 9044.947} C_VEL
LIN {X 0,Y 612.36,Z 838.971,A -85,B 0,C 180,E1 9050.991,E2 9050.991} C_VEL
LIN {X 0,Y 615.291,Z 849.461,A -85,B 0,C 180,E1 9051.567,E2 9051.567} C_VEL
LIN {X 0,Y 608.542,Z 919.872,A -85,B 0,C 180,E1 9053.822,E2 9053.822} C_VEL
LIN {X 0,Y 598.748,Z 990.522,A -85,B 0,C 180,E1 9057.592,E2 9057.592} C_VEL
LIN {X 0,Y 588.283,Z 1055.692,A -85,B 0,C 180,E1 9062.868,E2 9062.868} C_VEL
LIN {X 0,Y 579.484,Z 1111.501,A -85,B 0,C 180,E1 9069.461,E2 9069.461} C_VEL
LIN {X 0,Y 574.003,Z 1153.026,A -85,B 0,C 180,E1 9076.589,E2 9076.589} C_VEL
LIN {X 0,Y 571.671,Z 1179.774,A -85,B 0,C 180,E1 9083.486,E2 9083.486} C_VEL
LIN {X 0,Y 570.928,Z 1194.521,A -85,B 0,C 180,E1 9089.962,E2 9089.962} C_VEL
LIN {X 0,Y 570.794,Z 1199.98,A -85,B 0,C 180,E1 9096.832,E2 9096.832} C_VEL
LIN {X 0,Y 571.267,Z 1193.546,A -85,B 0,C 180,E1 9104.576,E2 9104.576} C_VEL
LIN {X 0,Y 572.697,Z 1172.734,A -85,B 0,C 180,E1 9112.551,E2 9112.551} C_VEL
LIN {X 0,Y 575.963,Z 1137.465,A -85,B 0,C 180,E1 9120.333,E2 9120.333} C_VEL
LIN {X 0,Y 582.915,Z 1088.815,A -85,B 0,C 180,E1 9127.434,E2 9127.434} C_VEL
LIN {X 0,Y 592.755,Z 1028.39,A -85,B 0,C 180,E1 9133.498,E2 9133.498} C_VEL
LIN {X 0,Y 603.147,Z 960.419,A -85,B 0,C 180,E1 9138.13,E2 9138.13} C_VEL
LIN {X 0,Y 611.852,Z 885.642,A -85,B 0,C 180,E1 9141.386,E2 9141.386} C_VEL
LIN {X 0,Y 614.543,Z 843.265,A -85,B 0,C 180,E1 9142.598,E2 9142.598} C_VEL
LIN {X 0,Y 580.967,Z 785.087,A -85,B 0,C 180,E1 9147.559,E2 9147.559} C_VEL
LIN {X 0,Y 570.164,Z 767.06,A -85,B 0,C 180,E1 9149.574,E2 9149.574} C_VEL
LIN {X 0,Y 570.292,Z 767.06,A -85,B 0,C 180,E1 9158.934,E2 9158.934} C_VEL
LIN {X 0,Y 571.183,Z 767.06,A -85,B 0,C 180,E1 9168.49,E2 9168.49} C_VEL
LIN {X 0,Y 571.231,Z 767.06,A -85,B 0,C 180,E1 9177.697,E2 9177.697} C_VEL
LIN {X 0,Y 570.524,Z 767.06,A -85,B 0,C 180,E1 9186.852,E2 9186.852} C_VEL
LIN {X 0,Y 570.358,Z 767.06,A -85,B 0,C 180,E1 9194.615,E2 9194.615} C_VEL
LIN {X 0,Y 569.964,Z 767.06,A -85,B 0,C 180,E1 9203.401,E2 9203.401} C_VEL
LIN {X 0,Y 569.978,Z 767.06,A -85,B 0,C 180,E1 9211.24,E2 9211.24} C_VEL
LIN {X 0,Y 570.024,Z 768.97,A -85,B 0,C 180,E1 9217.437,E2 9217.437} C_VEL
LIN {X 0,Y 607.769,Z 829.319,A -85,B 0,C 180,E1 9223.134,E2 9223.134} C_VEL
LIN {X 0,Y 615.972,Z 848.918,A -85,B 0,C 180,E1 9224.4,E2 9224.4} C_VEL
LIN {X 0,Y 608.875,Z 924.207,A -85,B 0,C 180,E1 9226.636,E2 9226.636} C_VEL
LIN {X 0,Y 602.207,Z 976.798,A -85,B 0,C 180,E1 9229.185,E2 9229.185} C_VEL
LIN {X 0,Y 591.282,Z 1007.222,A -85,B 0,C 180,E1 9230.587,E2 9230.587} C_VEL
LIN {X 0,Y 580.555,Z 1070.966,A -85,B 0,C 180,E1 9235.984,E2 9235.984} C_VEL
LIN {X 0,Y 571.556,Z 1125.565,A -85,B 0,C 180,E1 9242.718,E2 9242.718} C_VEL
LIN {X 0,Y 565.917,Z 1166.936,A -85,B 0,C 180,E1 9250.198,E2 9250.198} C_VEL
LIN {X 0,Y 563.444,Z 1193.384,A -85,B 0,C 180,E1 9257.598,E2 9257.598} C_VEL
LIN {X 0,Y 562.969,Z 1206.825,A -85,B 0,C 180,E1 9264.626,E2 9264.626} C_VEL
LIN {X 0,Y 562.644,Z 1209.829,A -85,B 0,C 180,E1 9270.811,E2 9270.811} C_VEL
LIN {X 0,Y 563.27,Z 1203.442,A -85,B 0,C 180,E1 9277.779,E2 9277.779} C_VEL
LIN {X 0,Y 564.746,Z 1183.357,A -85,B 0,C 180,E1 9285.624,E2 9285.624} C_VEL
LIN {X 0,Y 568.202,Z 1148.946,A -85,B 0,C 180,E1 9293.423,E2 9293.423} C_VEL
LIN {X 0,Y 575.285,Z 1101.581,A -85,B 0,C 180,E1 9300.554,E2 9300.554} C_VEL
LIN {X 0,Y 585.522,Z 1041.942,A -85,B 0,C 180,E1 9306.728,E2 9306.728} C_VEL
LIN {X 0,Y 596.195,Z 975.03,A -85,B 0,C 180,E1 9311.433,E2 9311.433} C_VEL
LIN {X 0,Y 605.541,Z 899.656,A -85,B 0,C 180,E1 9314.819,E2 9314.819} C_VEL
LIN {X 0,Y 609.058,Z 846.764,A -85,B 0,C 180,E1 9316.321,E2 9316.321} C_VEL
LIN {X 0,Y 573.25,Z 785.751,A -85,B 0,C 180,E1 9321.437,E2 9321.437} C_VEL
LIN {X 0,Y 562.099,Z 767.06,A -85,B 0,C 180,E1 9323.192,E2 9323.192} C_VEL
LIN {X 0,Y 562.408,Z 767.06,A -85,B 0,C 180,E1 9331.858,E2 9331.858} C_VEL
LIN {X 0,Y 562.06,Z 767.06,A -85,B 0,C 180,E1 9340.305,E2 9340.305} C_VEL
LIN {X 0,Y 562.583,Z 767.06,A -85,B 0,C 180,E1 9349.926,E2 9349.926} C_VEL
LIN {X 0,Y 563.388,Z 767.06,A -85,B 0,C 180,E1 9359.249,E2 9359.249} C_VEL
LIN {X 0,Y 562.547,Z 767.06,A -85,B 0,C 180,E1 9368.55,E2 9368.55} C_VEL
LIN {X 0,Y 562.261,Z 767.06,A -85,B 0,C 180,E1 9376.537,E2 9376.537} C_VEL
LIN {X 0,Y 562.07,Z 767.06,A -85,B 0,C 180,E1 9385.18,E2 9385.18} C_VEL
LIN {X 0,Y 561.923,Z 767.06,A -85,B 0,C 180,E1 9394.492,E2 9394.492} C_VEL
LIN {X 0,Y 561.957,Z 767.97,A -85,B 0,C 180,E1 9403.947,E2 9403.947} C_VEL
LIN {X 0,Y 605.757,Z 840.669,A -85,B 0,C 180,E1 9410.388,E2 9410.388} C_VEL
LIN {X 0,Y 609.334,Z 853.552,A -85,B 0,C 180,E1 9411.124,E2 9411.124} C_VEL
LIN {X 0,Y 602.083,Z 924.071,A -85,B 0,C 180,E1 9413.476,E2 9413.476} C_VEL
LIN {X 0,Y 591.686,Z 994.716,A -85,B 0,C 180,E1 9417.375,E2 9417.375} C_VEL
LIN {X 0,Y 580.741,Z 1059.129,A -85,B 0,C 180,E1 9422.751,E2 9422.751} C_VEL
LIN {X 0,Y 571.722,Z 1113.576,A -85,B 0,C 180,E1 9429.373,E2 9429.373} C_VEL
LIN {X 0,Y 565.933,Z 1155.346,A -85,B 0,C 180,E1 9436.788,E2 9436.788} C_VEL
LIN {X 0,Y 563.561,Z 1181.155,A -85,B 0,C 180,E1 9443.779,E2 9443.779} C_VEL
LIN {X 0,Y 562.932,Z 1194.668,A -85,B 0,C 180,E1 9449.962,E2 9449.962} C_VEL
LIN {X 0,Y 562.785,Z 1199.999,A -85,B 0,C 180,E1 9456.93,E2 9456.93} C_VEL
LIN {X 0,Y 563.288,Z 1193.375,A -85,B 0,C 180,E1 9464.787,E2 9464.787} C_VEL
LIN {X 0,Y 564.719,Z 1172.362,A -85,B 0,C 180,E1 9472.887,E2 9472.887} C_VEL
LIN {X 0,Y 568.247,Z 1137.459,A -85,B 0,C 180,E1 9480.67,E2 9480.67} C_VEL
LIN {X 0,Y 575.65,Z 1088.901,A -85,B 0,C 180,E1 9487.848,E2 9487.848} C_VEL
LIN {X 0,Y 586.012,Z 1028.584,A -85,B 0,C 180,E1 9493.969,E2 9493.969} C_VEL
LIN {X 0,Y 597.187,Z 959.81,A -85,B 0,C 180,E1 9498.68,E2 9498.68} C_VEL
LIN {X 0,Y 606.307,Z 884.205,A -85,B 0,C 180,E1 9501.968,E2 9501.968} C_VEL
LIN {X 0,Y 608.655,Z 846.65,A -85,B 0,C 180,E1 9503.072,E2 9503.072} C_VEL
LIN {X 0,Y 576.66,Z 790.376,A -85,B 0,C 180,E1 9508.011,E2 9508.011} C_VEL
LIN {X 0,Y 562.159,Z 767.06,A -85,B 0,C 180,E1 9510.666,E2 9510.666} C_VEL
LIN {X 0,Y 562.25,Z 767.06,A -85,B 0,C 180,E1 9520.269,E2 9520.269} C_VEL
LIN {X 0,Y 562.99,Z 767.06,A -85,B 0,C 180,E1 9529.426,E2 9529.426} C_VEL
LIN {X 0,Y 563.221,Z 767.06,A -85,B 0,C 180,E1 9537.664,E2 9537.664} C_VEL
LIN {X 0,Y 562.495,Z 767.06,A -85,B 0,C 180,E1 9546.95,E2 9546.95} C_VEL
LIN {X 0,Y 562.302,Z 767.06,A -85,B 0,C 180,E1 9554.829,E2 9554.829} C_VEL
LIN {X 0,Y 562.029,Z 767.06,A -85,B 0,C 180,E1 9563.017,E2 9563.017} C_VEL
LIN {X 0,Y 561.889,Z 767.06,A -85,B 0,C 180,E1 9571.796,E2 9571.796} C_VEL
LIN {X 0,Y 562.072,Z 768.939,A -85,B 0,C 180,E1 9576.279,E2 9576.279} C_VEL
LIN {X 0,Y 599.003,Z 827.166,A -85,B 0,C 180,E1 9582.187,E2 9582.187} C_VEL
LIN {X 0,Y 610.146,Z 852.024,A -85,B 0,C 180,E1 9583.924,E2 9583.924} C_VEL
LIN {X 0,Y 602.81,Z 925.35,A -85,B 0,C 180,E1 9586.154,E2 9586.154} C_VEL
LIN {X 0,Y 592.699,Z 997.64,A -85,B 0,C 180,E1 9589.944,E2 9589.944} C_VEL
LIN {X 0,Y 591.282,Z 1007.222,A -85,B 0,C 180,E1 9590.587,E2 9590.587} C_VEL
LIN {X 0,Y 579.855,Z 1036.082,A -85,B 0,C 180,E1 9592.274,E2 9592.274} C_VEL
LIN {X 0,Y 568.871,Z 1096.611,A -85,B 0,C 180,E1 9598.379,E2 9598.379} C_VEL
LIN {X 0,Y 560.918,Z 1144.865,A -85,B 0,C 180,E1 9605.467,E2 9605.467} C_VEL
LIN {X 0,Y 556.805,Z 1179.815,A -85,B 0,C 180,E1 9613.114,E2 9613.114} C_VEL
LIN {X 0,Y 555.499,Z 1200.675,A -85,B 0,C 180,E1 9620.607,E2 9620.607} C_VEL
LIN {X 0,Y 555.273,Z 1209.424,A -85,B 0,C 180,E1 9627.69,E2 9627.69} C_VEL
LIN {X 0,Y 555.032,Z 1206.738,A -85,B 0,C 180,E1 9635.529,E2 9635.529} C_VEL
LIN {X 0,Y 555.539,Z 1193.165,A -85,B 0,C 180,E1 9642.66,E2 9642.66} C_VEL
LIN {X 0,Y 558.183,Z 1166.505,A -85,B 0,C 180,E1 9650.189,E2 9650.189} C_VEL
LIN {X 0,Y 564.274,Z 1124.746,A -85,B 0,C 180,E1 9657.798,E2 9657.798} C_VEL
LIN {X 0,Y 573.59,Z 1070.978,A -85,B 0,C 180,E1 9664.486,E2 9664.486} C_VEL
LIN {X 0,Y 585.053,Z 1006.361,A -85,B 0,C 180,E1 9669.982,E2 9669.982} C_VEL
LIN {X 0,Y 595.812,Z 935.545,A -85,B 0,C 180,E1 9673.943,E2 9673.943} C_VEL
LIN {X 0,Y 603.486,Z 865.365,A -85,B 0,C 180,E1 9676.316,E2 9676.316} C_VEL
LIN {X 0,Y 603.166,Z 849.759,A -85,B 0,C 180,E1 9676.826,E2 9676.826} C_VEL
LIN {X 0,Y 568.076,Z 790.243,A -85,B 0,C 180,E1 9681.967,E2 9681.967} C_VEL
LIN {X 0,Y 554.091,Z 767.06,A -85,B 0,C 180,E1 9684.439,E2 9684.439} C_VEL
LIN {X 0,Y 554.397,Z 767.06,A -85,B 0,C 180,E1 9693.185,E2 9693.185} C_VEL
LIN {X 0,Y 554.328,Z 767.06,A -85,B 0,C 180,E1 9703.323,E2 9703.323} C_VEL
LIN {X 0,Y 554.543,Z 767.06,A -85,B 0,C 180,E1 9712.95,E2 9712.95} C_VEL
LIN {X 0,Y 554.743,Z 767.06,A -85,B 0,C 180,E1 9720.804,E2 9720.804} C_VEL
LIN {X 0,Y 554.513,Z 767.06,A -85,B 0,C 180,E1 9728.674,E2 9728.674} C_VEL
LIN {X 0,Y 554.241,Z 767.06,A -85,B 0,C 180,E1 9736.723,E2 9736.723} C_VEL
LIN {X 0,Y 554.089,Z 767.06,A -85,B 0,C 180,E1 9745.132,E2 9745.132} C_VEL
LIN {X 0,Y 553.911,Z 767.06,A -85,B 0,C 180,E1 9754.179,E2 9754.179} C_VEL
LIN {X 0,Y 554.095,Z 768.937,A -85,B 0,C 180,E1 9762.951,E2 9762.951} C_VEL
LIN {X 0,Y 598.023,Z 839.951,A -85,B 0,C 180,E1 9769.581,E2 9769.581} C_VEL
LIN {X 0,Y 603.636,Z 854.91,A -85,B 0,C 180,E1 9770.61,E2 9770.61} C_VEL
LIN {X 0,Y 596.142,Z 924.497,A -85,B 0,C 180,E1 9772.952,E2 9772.952} C_VEL
LIN {X 0,Y 585.332,Z 994.877,A -85,B 0,C 180,E1 9776.865,E2 9776.865} C_VEL
LIN {X 0,Y 573.648,Z 1060.292,A -85,B 0,C 180,E1 9782.402,E2 9782.402} C_VEL
LIN {X 0,Y 563.946,Z 1115.651,A -85,B 0,C 180,E1 9789.281,E2 9789.281} C_VEL
LIN {X 0,Y 558.119,Z 1155.828,A -85,B 0,C 180,E1 9796.6,E2 9796.6} C_VEL
LIN {X 0,Y 555.627,Z 1181.437,A -85,B 0,C 180,E1 9803.69,E2 9803.69} C_VEL
LIN {X 0,Y 554.944,Z 1194.816,A -85,B 0,C 180,E1 9809.961,E2 9809.961} C_VEL
LIN {X 0,Y 554.806,Z 1199.991,A -85,B 0,C 180,E1 9817.03,E2 9817.03} C_VEL
LIN {X 0,Y 555.328,Z 1193.205,A -85,B 0,C 180,E1 9825.004,E2 9825.004} C_VEL
LIN {X 0,Y 556.744,Z 1171.99,A -85,B 0,C 180,E1 9833.234,E2 9833.234} C_VEL
LIN {X 0,Y 560.526,Z 1137.646,A -85,B 0,C 180,E1 9840.982,E2 9840.982} C_VEL
LIN {X 0,Y 568.197,Z 1090.503,A -85,B 0,C 180,E1 9848.086,E2 9848.086} C_VEL
LIN {X 0,Y 579.037,Z 1030.598,A -85,B 0,C 180,E1 9854.293,E2 9854.293} C_VEL
LIN {X 0,Y 590.637,Z 962.584,A -85,B 0,C 180,E1 9859.061,E2 9859.061} C_VEL
LIN {X 0,Y 600.283,Z 887.016,A -85,B 0,C 180,E1 9862.424,E2 9862.424} C_VEL
LIN {X 0,Y 602.826,Z 850.038,A -85,B 0,C 180,E1 9863.542,E2 9863.542} C_VEL
LIN {X 0,Y 570.988,Z 793.029,A -85,B 0,C 180,E1 9868.719,E2 9868.719} C_VEL
LIN {X 0,Y 554.098,Z 767.06,A -85,B 0,C 180,E1 9872.106,E2 9872.106} C_VEL
LIN {X 0,Y 554.259,Z 767.06,A -85,B 0,C 180,E1 9881.633,E2 9881.633} C_VEL
LIN {X 0,Y 554.963,Z 767.06,A -85,B 0,C 180,E1 9889.745,E2 9889.745} C_VEL
LIN {X 0,Y 554.648,Z 767.06,A -85,B 0,C 180,E1 9899.196,E2 9899.196} C_VEL
LIN {X 0,Y 554.487,Z 767.06,A -85,B 0,C 180,E1 9907.051,E2 9907.051} C_VEL
LIN {X 0,Y 554.252,Z 767.06,A -85,B 0,C 180,E1 9915.049,E2 9915.049} C_VEL
LIN {X 0,Y 553.933,Z 767.06,A -85,B 0,C 180,E1 9923.52,E2 9923.52} C_VEL
LIN {X 0,Y 553.845,Z 767.06,A -85,B 0,C 180,E1 9932.258,E2 9932.258} C_VEL
LIN {X 0,Y 554.037,Z 768.998,A -85,B 0,C 180,E1 9935.033,E2 9935.033} C_VEL
LIN {X 0,Y 589.739,Z 823.958,A -85,B 0,C 180,E1 9941.086,E2 9941.086} C_VEL
LIN {X 0,Y 604.375,Z 855.104,A -85,B 0,C 180,E1 9943.44,E2 9943.44} C_VEL
LIN {X 0,Y 596.55,Z 928.877,A -85,B 0,C 180,E1 9945.765,E2 9945.765} C_VEL
LIN {X 0,Y 585.61,Z 1002.396,A -85,B 0,C 180,E1 9949.744,E2 9949.744} C_VEL
LIN {X 0,Y 579.855,Z 1036.082,A -85,B 0,C 180,E1 9952.274,E2 9952.274} C_VEL
LIN {X 0,Y 568.22,Z 1063.176,A -85,B 0,C 180,E1 9954.252,E2 9954.252} C_VEL
LIN {X 0,Y 558.045,Z 1118.534,A -85,B 0,C 180,E1 9960.893,E2 9960.893} C_VEL
LIN {X 0,Y 551.44,Z 1161.791,A -85,B 0,C 180,E1 9968.487,E2 9968.487} C_VEL
LIN {X 0,Y 547.914,Z 1191.109,A -85,B 0,C 180,E1 9976.426,E2 9976.426} C_VEL
LIN {X 0,Y 547.082,Z 1205.925,A -85,B 0,C 180,E1 9983.67,E2 9983.67} C_VEL
LIN {X 0,Y 546.764,Z 1209.846,A -85,B 0,C 180,E1 9989.244,E2 9989.244} C_VEL
LIN {X 0,Y 547.041,Z 1205.826,A -85,B 0,C 180,E1 9996.409,E2 9996.409} C_VEL
LIN {X 0,Y 548.135,Z 1189.393,A -85,B 0,C 180,E1 10004.178,E2 10004.178} C_VEL
LIN {X 0,Y 551.982,Z 1157.265,A -85,B 0,C 180,E1 10012.474,E2 10012.474} C_VEL
LIN {X 0,Y 559.349,Z 1111.12,A -85,B 0,C 180,E1 10020.165,E2 10020.165} C_VEL
LIN {X 0,Y 569.942,Z 1054.286,A -85,B 0,C 180,E1 10026.62,E2 10026.62} C_VEL
LIN {X 0,Y 581.739,Z 987.876,A -85,B 0,C 180,E1 10031.738,E2 10031.738} C_VEL
LIN {X 0,Y 592.807,Z 912.227,A -85,B 0,C 180,E1 10035.456,E2 10035.456} C_VEL
LIN {X 0,Y 597.481,Z 853.223,A -85,B 0,C 180,E1 10037.312,E2 10037.312} C_VEL
LIN {X 0,Y 561.569,Z 792.002,A -85,B 0,C 180,E1 10042.73,E2 10042.73} C_VEL
LIN {X 0,Y 546.092,Z 767.06,A -85,B 0,C 180,E1 10045.313,E2 10045.313} C_VEL
LIN {X 0,Y 546.377,Z 767.06,A -85,B 0,C 180,E1 10054.582,E2 10054.582} C_VEL
LIN {X 0,Y 546.279,Z 767.06,A -85,B 0,C 180,E1 10064.726,E2 10064.726} C_VEL
LIN {X 0,Y 546.542,Z 767.06,A -85,B 0,C 180,E1 10072.846,E2 10072.846} C_VEL
LIN {X 0,Y 546.748,Z 767.06,A -85,B 0,C 180,E1 10080.816,E2 10080.816} C_VEL
LIN {X 0,Y 546.361,Z 767.06,A -85,B 0,C 180,E1 10089.412,E2 10089.412} C_VEL
LIN {X 0,Y 546.049,Z 767.06,A -85,B 0,C 180,E1 10098.653,E2 10098.653} C_VEL
LIN {X 0,Y 546.003,Z 767.06,A -85,B 0,C 180,E1 10107.308,E2 10107.308} C_VEL
LIN {X 0,Y 545.878,Z 767.06,A -85,B 0,C 180,E1 10116.715,E2 10116.715} C_VEL
LIN {X 0,Y 546.073,Z 768.766,A -85,B 0,C 180,E1 10121.861,E2 10121.861} C_VEL
LIN {X 0,Y 591.365,Z 841.502,A -85,B 0,C 180,E1 10128.925,E2 10128.925} C_VEL
LIN {X 0,Y 597.798,Z 858.093,A -85,B 0,C 180,E1 10130.128,E2 10130.128} C_VEL
LIN {X 0,Y 589.746,Z 928.599,A -85,B 0,C 180,E1 10132.584,E2 10132.584} C_VEL
LIN {X 0,Y 578.535,Z 997.777,A -85,B 0,C 180,E1 10136.537,E2 10136.537} C_VEL
LIN {X 0,Y 566.387,Z 1062.345,A -85,B 0,C 180,E1 10142.134,E2 10142.134} C_VEL
LIN {X 0,Y 556.435,Z 1116.369,A -85,B 0,C 180,E1 10148.988,E2 10148.988} C_VEL
LIN {X 0,Y 550.315,Z 1156.308,A -85,B 0,C 180,E1 10156.406,E2 10156.406} C_VEL
LIN {X 0,Y 547.677,Z 1181.72,A -85,B 0,C 180,E1 10163.598,E2 10163.598} C_VEL
LIN {X 0,Y 546.958,Z 1194.964,A -85,B 0,C 180,E1 10169.961,E2 10169.961} C_VEL
LIN {X 0,Y 546.796,Z 1199.97,A -85,B 0,C 180,E1 10177.134,E2 10177.134} C_VEL
LIN {X 0,Y 547.341,Z 1193.033,A -85,B 0,C 180,E1 10185.228,E2 10185.228} C_VEL
LIN {X 0,Y 548.795,Z 1171.593,A -85,B 0,C 180,E1 10193.591,E2 10193.591} C_VEL
LIN {X 0,Y 552.789,Z 1138.313,A -85,B 0,C 180,E1 10201.212,E2 10201.212} C_VEL
LIN {X 0,Y 561.003,Z 1090.268,A -85,B 0,C 180,E1 10208.562,E2 10208.562} C_VEL
LIN {X 0,Y 572.538,Z 1030.179,A -85,B 0,C 180,E1 10214.838,E2 10214.838} C_VEL
LIN {X 0,Y 584.665,Z 962.346,A -85,B 0,C 180,E1 10219.615,E2 10219.615} C_VEL
LIN {X 0,Y 594.726,Z 886.595,A -85,B 0,C 180,E1 10222.993,E2 10222.993} C_VEL
LIN {X 0,Y 596.877,Z 853.07,A -85,B 0,C 180,E1 10224.048,E2 10224.048} C_VEL
LIN {X 0,Y 567.022,Z 798.809,A -85,B 0,C 180,E1 10229.147,E2 10229.147} C_VEL
LIN {X 0,Y 546.069,Z 767.06,A -85,B 0,C 180,E1 10233.142,E2 10233.142} C_VEL
LIN {X 0,Y 546.257,Z 767.06,A -85,B 0,C 180,E1 10241.354,E2 10241.354} C_VEL
LIN {X 0,Y 546.971,Z 767.06,A -85,B 0,C 180,E1 10249.759,E2 10249.759} C_VEL
LIN {X 0,Y 546.659,Z 767.06,A -85,B 0,C 180,E1 10259.184,E2 10259.184} C_VEL
LIN {X 0,Y 546.46,Z 767.06,A -85,B 0,C 180,E1 10267.155,E2 10267.155} C_VEL
LIN {X 0,Y 546.204,Z 767.06,A -85,B 0,C 180,E1 10275.276,E2 10275.276} C_VEL
LIN {X 0,Y 545.909,Z 767.06,A -85,B 0,C 180,E1 10283.738,E2 10283.738} C_VEL
LIN {X 0,Y 545.868,Z 767.06,A -85,B 0,C 180,E1 10293.368,E2 10293.368} C_VEL
LIN {X 0,Y 579.243,Z 818.923,A -85,B 0,C 180,E1 10299.704,E2 10299.704} C_VEL
LIN {X 0,Y 598.644,Z 857.571,A -85,B 0,C 180,E1 10302.943,E2 10302.943} C_VEL
LIN {X 0,Y 590.281,Z 932.876,A -85,B 0,C 180,E1 10305.39,E2 10305.39} C_VEL
LIN {X 0,Y 578.841,Z 1005.048,A -85,B 0,C 180,E1 10309.398,E2 10309.398} C_VEL
LIN {X 0,Y 568.22,Z 1063.176,A -85,B 0,C 180,E1 10314.252,E2 10314.252} C_VEL
LIN {X 0,Y 556.224,Z 1088.426,A -85,B 0,C 180,E1 10316.489,E2 10316.489} C_VEL
LIN {X 0,Y 546.85,Z 1138.843,A -85,B 0,C 180,E1 10323.69,E2 10323.69} C_VEL
LIN {X 0,Y 541.437,Z 1174.802,A -85,B 0,C 180,E1 10331.242,E2 10331.242} C_VEL
LIN {X 0,Y 539.331,Z 1197.292,A -85,B 0,C 180,E1 10338.683,E2 10338.683} C_VEL
LIN {X 0,Y 539.267,Z 1208.401,A -85,B 0,C 180,E1 10346.006,E2 10346.006} C_VEL
LIN {X 0,Y 539.307,Z 1208.343,A -85,B 0,C 180,E1 10354.073,E2 10354.073} C_VEL
LIN {X 0,Y 539.45,Z 1197.102,A -85,B 0,C 180,E1 10361.395,E2 10361.395} C_VEL
LIN {X 0,Y 541.495,Z 1174.494,A -85,B 0,C 180,E1 10368.84,E2 10368.84} C_VEL
LIN {X 0,Y 547.044,Z 1137.156,A -85,B 0,C 180,E1 10376.611,E2 10376.611} C_VEL
LIN {X 0,Y 556.667,Z 1085.881,A -85,B 0,C 180,E1 10383.821,E2 10383.821} C_VEL
LIN {X 0,Y 569.041,Z 1023.918,A -85,B 0,C 180,E1 10389.732,E2 10389.732} C_VEL
LIN {X 0,Y 581.109,Z 955.644,A -85,B 0,C 180,E1 10394.08,E2 10394.08} C_VEL
LIN {X 0,Y 590.615,Z 882.825,A -85,B 0,C 180,E1 10396.977,E2 10396.977} C_VEL
LIN {X 0,Y 591.659,Z 856.269,A -85,B 0,C 180,E1 10397.826,E2 10397.826} C_VEL
LIN {X 0,Y 555.649,Z 795.122,A -85,B 0,C 180,E1 10403.417,E2 10403.417} C_VEL
LIN {X 0,Y 538.072,Z 767.06,A -85,B 0,C 180,E1 10406.676,E2 10406.676} C_VEL
LIN {X 0,Y 538.272,Z 767.06,A -85,B 0,C 180,E1 10415.904,E2 10415.904} C_VEL
LIN {X 0,Y 538.25,Z 767.06,A -85,B 0,C 180,E1 10426.162,E2 10426.162} C_VEL
LIN {X 0,Y 538.38,Z 767.06,A -85,B 0,C 180,E1 10434.362,E2 10434.362} C_VEL
LIN {X 0,Y 538.74,Z 767.06,A -85,B 0,C 180,E1 10440.828,E2 10440.828} C_VEL
LIN {X 0,Y 538.46,Z 767.06,A -85,B 0,C 180,E1 10448.935,E2 10448.935} C_VEL
LIN {X 0,Y 538.144,Z 767.06,A -85,B 0,C 180,E1 10457.239,E2 10457.239} C_VEL
LIN {X 0,Y 537.983,Z 767.06,A -85,B 0,C 180,E1 10465.94,E2 10465.94} C_VEL
LIN {X 0,Y 537.825,Z 767.06,A -85,B 0,C 180,E1 10475.351,E2 10475.351} C_VEL
LIN {X 0,Y 538.028,Z 768.584,A -85,B 0,C 180,E1 10480.71,E2 10480.71} C_VEL
LIN {X 0,Y 583.845,Z 841.425,A -85,B 0,C 180,E1 10488.117,E2 10488.117} C_VEL
LIN {X 0,Y 591.937,Z 861.994,A -85,B 0,C 180,E1 10489.655,E2 10489.655} C_VEL
LIN {X 0,Y 583.209,Z 933.701,A -85,B 0,C 180,E1 10492.265,E2 10492.265} C_VEL
LIN {X 0,Y 571.239,Z 1003.336,A -85,B 0,C 180,E1 10496.396,E2 10496.396} C_VEL
LIN {X 0,Y 558.558,Z 1067.096,A -85,B 0,C 180,E1 10502.145,E2 10502.145} C_VEL
LIN {X 0,Y 548.112,Z 1120.827,A -85,B 0,C 180,E1 10509.291,E2 10509.291} C_VEL
LIN {X 0,Y 541.913,Z 1160.119,A -85,B 0,C 180,E1 10517.016,E2 10517.016} C_VEL
LIN {X 0,Y 539.54,Z 1184.186,A -85,B 0,C 180,E1 10524.312,E2 10524.312} C_VEL
LIN {X 0,Y 538.866,Z 1196.216,A -85,B 0,C 180,E1 10530.767,E2 10530.767} C_VEL
LIN {X 0,Y 538.786,Z 1199.948,A -85,B 0,C 180,E1 10537.24,E2 10537.24} C_VEL
LIN {X 0,Y 539.236,Z 1194.122,A -85,B 0,C 180,E1 10544.628,E2 10544.628} C_VEL
LIN {X 0,Y 540.827,Z 1174.056,A -85,B 0,C 180,E1 10553.084,E2 10553.084} C_VEL
LIN {X 0,Y 544.934,Z 1140.167,A -85,B 0,C 180,E1 10561.212,E2 10561.212} C_VEL
LIN {X 0,Y 553.31,Z 1093.646,A -85,B 0,C 180,E1 10568.582,E2 10568.582} C_VEL
LIN {X 0,Y 565.273,Z 1034.121,A -85,B 0,C 180,E1 10575.02,E2 10575.02} C_VEL
LIN {X 0,Y 577.984,Z 966.073,A -85,B 0,C 180,E1 10579.957,E2 10579.957} C_VEL
LIN {X 0,Y 588.584,Z 891.115,A -85,B 0,C 180,E1 10583.405,E2 10583.405} C_VEL
LIN {X 0,Y 591.143,Z 856.459,A -85,B 0,C 180,E1 10584.544,E2 10584.544} C_VEL
LIN {X 0,Y 562.866,Z 804.189,A -85,B 0,C 180,E1 10589.624,E2 10589.624} C_VEL
LIN {X 0,Y 538.101,Z 767.06,A -85,B 0,C 180,E1 10594.761,E2 10594.761} C_VEL
LIN {X 0,Y 538.638,Z 767.06,A -85,B 0,C 180,E1 10604.46,E2 10604.46} C_VEL
LIN {X 0,Y 538.42,Z 767.06,A -85,B 0,C 180,E1 10612.695,E2 10612.695} C_VEL
LIN {X 0,Y 538.66,Z 767.06,A -85,B 0,C 180,E1 10619.172,E2 10619.172} C_VEL
LIN {X 0,Y 538.435,Z 767.06,A -85,B 0,C 180,E1 10627.262,E2 10627.262} C_VEL
LIN {X 0,Y 538.171,Z 767.06,A -85,B 0,C 180,E1 10635.51,E2 10635.51} C_VEL
LIN {X 0,Y 537.86,Z 767.06,A -85,B 0,C 180,E1 10644.116,E2 10644.116} C_VEL
LIN {X 0,Y 538.079,Z 768.97,A -85,B 0,C 180,E1 10652.277,E2 10652.277} C_VEL
LIN {X 0,Y 571.72,Z 818.705,A -85,B 0,C 180,E1 10658.724,E2 10658.724} C_VEL
LIN {X 0,Y 592.896,Z 860.94,A -85,B 0,C 180,E1 10662.455,E2 10662.455} C_VEL
LIN {X 0,Y 584.092,Z 935.273,A -85,B 0,C 180,E1 10664.943,E2 10664.943} C_VEL
LIN {X 0,Y 571.987,Z 1007.834,A -85,B 0,C 180,E1 10669.068,E2 10669.068} C_VEL
LIN {X 0,Y 559.779,Z 1071.808,A -85,B 0,C 180,E1 10674.641,E2 10674.641} C_VEL
LIN {X 0,Y 556.224,Z 1088.426,A -85,B 0,C 180,E1 10676.489,E2 10676.489} C_VEL
LIN {X 0,Y 544.613,Z 1111.638,A -85,B 0,C 180,E1 10679.012,E2 10679.012} C_VEL
LIN {X 0,Y 536.516,Z 1157.151,A -85,B 0,C 180,E1 10686.815,E2 10686.815} C_VEL
LIN {X 0,Y 532.557,Z 1188.978,A -85,B 0,C 180,E1 10695.249,E2 10695.249} C_VEL
LIN {X 0,Y 531.123,Z 1205.925,A -85,B 0,C 180,E1 10703.479,E2 10703.479} C_VEL
LIN {X 0,Y 530.783,Z 1209.845,A -85,B 0,C 180,E1 10709.221,E2 10709.221} C_VEL
LIN {X 0,Y 531.091,Z 1205.826,A -85,B 0,C 180,E1 10716.602,E2 10716.602} C_VEL
LIN {X 0,Y 532.44,Z 1189.118,A -85,B 0,C 180,E1 10724.704,E2 10724.704} C_VEL
LIN {X 0,Y 536.425,Z 1158.38,A -85,B 0,C 180,E1 10732.911,E2 10732.911} C_VEL
LIN {X 0,Y 544.314,Z 1113.862,A -85,B 0,C 180,E1 10740.653,E2 10740.653} C_VEL
LIN {X 0,Y 555.89,Z 1057.38,A -85,B 0,C 180,E1 10747.32,E2 10747.32} C_VEL
LIN {X 0,Y 568.913,Z 990.746,A -85,B 0,C 180,E1 10752.641,E2 10752.641} C_VEL
LIN {X 0,Y 580.942,Z 916.214,A -85,B 0,C 180,E1 10756.433,E2 10756.433} C_VEL
LIN {X 0,Y 586.096,Z 860.107,A -85,B 0,C 180,E1 10758.279,E2 10758.279} C_VEL
LIN {X 0,Y 549.769,Z 797.928,A -85,B 0,C 180,E1 10764.128,E2 10764.128} C_VEL
LIN {X 0,Y 530.103,Z 767.06,A -85,B 0,C 180,E1 10767.678,E2 10767.678} C_VEL
LIN {X 0,Y 530.109,Z 767.06,A -85,B 0,C 180,E1 10777.298,E2 10777.298} C_VEL
LIN {X 0,Y 530.228,Z 767.06,A -85,B 0,C 180,E1 10785.948,E2 10785.948} C_VEL
LIN {X 0,Y 530.38,Z 767.06,A -85,B 0,C 180,E1 10794.276,E2 10794.276} C_VEL
LIN {X 0,Y 530.733,Z 767.06,A -85,B 0,C 180,E1 10800.84,E2 10800.84} C_VEL
LIN {X 0,Y 530.429,Z 767.06,A -85,B 0,C 180,E1 10809.072,E2 10809.072} C_VEL
LIN {X 0,Y 530.102,Z 767.06,A -85,B 0,C 180,E1 10817.508,E2 10817.508} C_VEL
LIN {X 0,Y 529.979,Z 767.06,A -85,B 0,C 180,E1 10826.361,E2 10826.361} C_VEL
LIN {X 0,Y 529.84,Z 767.06,A -85,B 0,C 180,E1 10835.965,E2 10835.965} C_VEL
LIN {X 0,Y 530.136,Z 768.965,A -85,B 0,C 180,E1 10839.531,E2 10839.531} C_VEL
LIN {X 0,Y 572.997,Z 835.874,A -85,B 0,C 180,E1 10846.751,E2 10846.751} C_VEL
LIN {X 0,Y 586.165,Z 865.431,A -85,B 0,C 180,E1 10849.167,E2 10849.167} C_VEL
LIN {X 0,Y 576.947,Z 936.98,A -85,B 0,C 180,E1 10851.85,E2 10851.85} C_VEL
LIN {X 0,Y 564.71,Z 1004.765,A -85,B 0,C 180,E1 10855.954,E2 10855.954} C_VEL
LIN {X 0,Y 551.504,Z 1068.106,A -85,B 0,C 180,E1 10861.757,E2 10861.757} C_VEL
LIN {X 0,Y 540.612,Z 1121.479,A -85,B 0,C 180,E1 10868.99,E2 10868.99} C_VEL
LIN {X 0,Y 534.085,Z 1160.548,A -85,B 0,C 180,E1 10876.822,E2 10876.822} C_VEL
LIN {X 0,Y 531.564,Z 1184.448,A -85,B 0,C 180,E1 10884.226,E2 10884.226} C_VEL
LIN {X 0,Y 530.893,Z 1196.337,A -85,B 0,C 180,E1 10890.778,E2 10890.778} C_VEL
LIN {X 0,Y 530.777,Z 1199.927,A -85,B 0,C 180,E1 10897.35,E2 10897.35} C_VEL
LIN {X 0,Y 531.281,Z 1193.965,A -85,B 0,C 180,E1 10904.852,E2 10904.852} C_VEL
LIN {X 0,Y 532.87,Z 1173.694,A -85,B 0,C 180,E1 10913.449,E2 10913.449} C_VEL
LIN {X 0,Y 537.203,Z 1140.78,A -85,B 0,C 180,E1 10921.454,E2 10921.454} C_VEL
LIN {X 0,Y 545.957,Z 1094.511,A -85,B 0,C 180,E1 10928.927,E2 10928.927} C_VEL
LIN {X 0,Y 558.5,Z 1035.276,A -85,B 0,C 180,E1 10935.449,E2 10935.449} C_VEL
LIN {X 0,Y 571.578,Z 968.277,A -85,B 0,C 180,E1 10940.392,E2 10940.392} C_VEL
LIN {X 0,Y 582.841,Z 893.186,A -85,B 0,C 180,E1 10943.916,E2 10943.916} C_VEL
LIN {X 0,Y 585.451,Z 859.685,A -85,B 0,C 180,E1 10945.065,E2 10945.065} C_VEL
LIN {X 0,Y 557.62,Z 807.568,A -85,B 0,C 180,E1 10950.322,E2 10950.322} C_VEL
LIN {X 0,Y 530.201,Z 767.06,A -85,B 0,C 180,E1 10956.304,E2 10956.304} C_VEL
LIN {X 0,Y 530.909,Z 767.06,A -85,B 0,C 180,E1 10965.922,E2 10965.922} C_VEL
LIN {X 0,Y 530.939,Z 767.06,A -85,B 0,C 180,E1 10975.882,E2 10975.882} C_VEL
LIN {X 0,Y 530.825,Z 767.06,A -85,B 0,C 180,E1 10985.719,E2 10985.719} C_VEL
LIN {X 0,Y 530.13,Z 767.06,A -85,B 0,C 180,E1 10995.751,E2 10995.751} C_VEL
LIN {X 0,Y 529.805,Z 767.06,A -85,B 0,C 180,E1 11004.506,E2 11004.506} C_VEL
LIN {X 0,Y 530.11,Z 768.911,A -85,B 0,C 180,E1 11010.732,E2 11010.732} C_VEL
LIN {X 0,Y 564.061,Z 818.192,A -85,B 0,C 180,E1 11017.66,E2 11017.66} C_VEL
LIN {X 0,Y 587.336,Z 863.616,A -85,B 0,C 180,E1 11021.94,E2 11021.94} C_VEL
LIN {X 0,Y 578.057,Z 937.046,A -85,B 0,C 180,E1 11024.456,E2 11024.456} C_VEL
LIN {X 0,Y 565.482,Z 1009.024,A -85,B 0,C 180,E1 11028.614,E2 11028.614} C_VEL
LIN {X 0,Y 552.509,Z 1073.697,A -85,B 0,C 180,E1 11034.355,E2 11034.355} C_VEL
LIN {X 0,Y 544.613,Z 1111.638,A -85,B 0,C 180,E1 11039.012,E2 11039.012} C_VEL
LIN {X 0,Y 533.237,Z 1132.666,A -85,B 0,C 180,E1 11041.818,E2 11041.818} C_VEL
LIN {X 0,Y 526.277,Z 1172.239,A -85,B 0,C 180,E1 11049.983,E2 11049.983} C_VEL
LIN {X 0,Y 523.54,Z 1195.356,A -85,B 0,C 180,E1 11057.488,E2 11057.488} C_VEL
LIN {X 0,Y 523.028,Z 1206.81,A -85,B 0,C 180,E1 11064.214,E2 11064.214} C_VEL
LIN {X 0,Y 522.7,Z 1209.828,A -85,B 0,C 180,E1 11070.873,E2 11070.873} C_VEL
LIN {X 0,Y 523.44,Z 1203.427,A -85,B 0,C 180,E1 11078.375,E2 11078.375} C_VEL
LIN {X 0,Y 525.1,Z 1183.352,A -85,B 0,C 180,E1 11086.838,E2 11086.838} C_VEL
LIN {X 0,Y 529.613,Z 1150.63,A -85,B 0,C 180,E1 11094.892,E2 11094.892} C_VEL
LIN {X 0,Y 538.875,Z 1104.202,A -85,B 0,C 180,E1 11102.471,E2 11102.471} C_VEL
LIN {X 0,Y 552,Z 1044.146,A -85,B 0,C 180,E1 11109.088,E2 11109.088} C_VEL
LIN {X 0,Y 565.474,Z 977.277,A -85,B 0,C 180,E1 11114.022,E2 11114.022} C_VEL
LIN {X 0,Y 576.924,Z 902.513,A -85,B 0,C 180,E1 11117.527,E2 11117.527} C_VEL
LIN {X 0,Y 580.319,Z 863.304,A -85,B 0,C 180,E1 11118.785,E2 11118.785} C_VEL
LIN {X 0,Y 542.972,Z 799.138,A -85,B 0,C 180,E1 11125.024,E2 11125.024} C_VEL
LIN {X 0,Y 522.12,Z 767.06,A -85,B 0,C 180,E1 11129.091,E2 11129.091} C_VEL
LIN {X 0,Y 522.026,Z 767.06,A -85,B 0,C 180,E1 11138.724,E2 11138.724} C_VEL
LIN {X 0,Y 522.223,Z 767.06,A -85,B 0,C 180,E1 11147.439,E2 11147.439} C_VEL
LIN {X 0,Y 522.367,Z 767.06,A -85,B 0,C 180,E1 11155.859,E2 11155.859} C_VEL
LIN {X 0,Y 522.463,Z 767.06,A -85,B 0,C 180,E1 11162.518,E2 11162.518} C_VEL
LIN {X 0,Y 522.223,Z 767.06,A -85,B 0,C 180,E1 11170.906,E2 11170.906} C_VEL
LIN {X 0,Y 522.002,Z 767.06,A -85,B 0,C 180,E1 11179.547,E2 11179.547} C_VEL
LIN {X 0,Y 521.92,Z 767.06,A -85,B 0,C 180,E1 11188.682,E2 11188.682} C_VEL
LIN {X 0,Y 522.09,Z 768.942,A -85,B 0,C 180,E1 11198.25,E2 11198.25} C_VEL
LIN {X 0,Y 563.716,Z 832.983,A -85,B 0,C 180,E1 11205.58,E2 11205.58} C_VEL
LIN {X 0,Y 580.38,Z 868.335,A -85,B 0,C 180,E1 11208.666,E2 11208.666} C_VEL
LIN {X 0,Y 570.677,Z 940.377,A -85,B 0,C 180,E1 11211.43,E2 11211.43} C_VEL
LIN {X 0,Y 557.668,Z 1008.844,A -85,B 0,C 180,E1 11215.7,E2 11215.7} C_VEL
LIN {X 0,Y 543.903,Z 1071.611,A -85,B 0,C 180,E1 11221.648,E2 11221.648} C_VEL
LIN {X 0,Y 532.539,Z 1124.609,A -85,B 0,C 180,E1 11229.094,E2 11229.094} C_VEL
LIN {X 0,Y 526.286,Z 1160.977,A -85,B 0,C 180,E1 11236.623,E2 11236.623} C_VEL
LIN {X 0,Y 523.613,Z 1184.708,A -85,B 0,C 180,E1 11244.138,E2 11244.138} C_VEL
LIN {X 0,Y 522.906,Z 1196.446,A -85,B 0,C 180,E1 11250.79,E2 11250.79} C_VEL
LIN {X 0,Y 522.783,Z 1199.905,A -85,B 0,C 180,E1 11257.463,E2 11257.463} C_VEL
LIN {X 0,Y 523.305,Z 1193.807,A -85,B 0,C 180,E1 11265.084,E2 11265.084} C_VEL
LIN {X 0,Y 524.947,Z 1173.769,A -85,B 0,C 180,E1 11273.679,E2 11273.679} C_VEL
LIN {X 0,Y 529.447,Z 1141.483,A -85,B 0,C 180,E1 11281.685,E2 11281.685} C_VEL
LIN {X 0,Y 538.663,Z 1095.405,A -85,B 0,C 180,E1 11289.277,E2 11289.277} C_VEL
LIN {X 0,Y 551.694,Z 1036.746,A -85,B 0,C 180,E1 11295.856,E2 11295.856} C_VEL
LIN {X 0,Y 565.448,Z 969.501,A -85,B 0,C 180,E1 11300.891,E2 11300.891} C_VEL
LIN {X 0,Y 577.206,Z 895.081,A -85,B 0,C 180,E1 11304.447,E2 11304.447} C_VEL
LIN {X 0,Y 580.066,Z 863.574,A -85,B 0,C 180,E1 11305.548,E2 11305.548} C_VEL
LIN {X 0,Y 553.271,Z 812.445,A -85,B 0,C 180,E1 11310.855,E2 11310.855} C_VEL
LIN {X 0,Y 523.981,Z 772.131,A -85,B 0,C 180,E1 11317.248,E2 11317.248} C_VEL
LIN {X 0,Y 522.129,Z 767.06,A -85,B 0,C 180,E1 11317.998,E2 11317.998} C_VEL
LIN {X 0,Y 523.003,Z 767.06,A -85,B 0,C 180,E1 11327.413,E2 11327.413} C_VEL
LIN {X 0,Y 523.225,Z 767.06,A -85,B 0,C 180,E1 11337.486,E2 11337.486} C_VEL
LIN {X 0,Y 522.792,Z 767.06,A -85,B 0,C 180,E1 11345.807,E2 11345.807} C_VEL
LIN {X 0,Y 522.306,Z 767.06,A -85,B 0,C 180,E1 11354.27,E2 11354.27} C_VEL
LIN {X 0,Y 521.807,Z 767.06,A -85,B 0,C 180,E1 11363.763,E2 11363.763} C_VEL
LIN {X 0,Y 522.055,Z 768.914,A -85,B 0,C 180,E1 11369.029,E2 11369.029} C_VEL
LIN {X 0,Y 554.131,Z 814.276,A -85,B 0,C 180,E1 11376.096,E2 11376.096} C_VEL
LIN {X 0,Y 581.751,Z 865.918,A -85,B 0,C 180,E1 11381.387,E2 11381.387} C_VEL
LIN {X 0,Y 572.32,Z 937.575,A -85,B 0,C 180,E1 11383.896,E2 11383.896} C_VEL
LIN {X 0,Y 559.036,Z 1010.067,A -85,B 0,C 180,E1 11388.139,E2 11388.139} C_VEL
LIN {X 0,Y 545.788,Z 1073.013,A -85,B 0,C 180,E1 11393.775,E2 11393.775} C_VEL
LIN {X 0,Y 534.853,Z 1125.325,A -85,B 0,C 180,E1 11400.631,E2 11400.631} C_VEL
LIN {X 0,Y 533.237,Z 1132.666,A -85,B 0,C 180,E1 11401.818,E2 11401.818} C_VEL
LIN {X 0,Y 521.897,Z 1151.337,A -85,B 0,C 180,E1 11404.863,E2 11404.863} C_VEL
LIN {X 0,Y 517.05,Z 1183.966,A -85,B 0,C 180,E1 11413.095,E2 11413.095} C_VEL
LIN {X 0,Y 515.497,Z 1203.543,A -85,B 0,C 180,E1 11421.579,E2 11421.579} C_VEL
LIN {X 0,Y 514.801,Z 1209.845,A -85,B 0,C 180,E1 11429.197,E2 11429.197} C_VEL
LIN {X 0,Y 515.12,Z 1205.826,A -85,B 0,C 180,E1 11436.808,E2 11436.808} C_VEL
LIN {X 0,Y 516.754,Z 1188.572,A -85,B 0,C 180,E1 11445.366,E2 11445.366} C_VEL
LIN {X 0,Y 521.072,Z 1157.807,A -85,B 0,C 180,E1 11453.759,E2 11453.759} C_VEL
LIN {X 0,Y 530.022,Z 1112.941,A -85,B 0,C 180,E1 11461.713,E2 11461.713} C_VEL
LIN {X 0,Y 543.074,Z 1055.273,A -85,B 0,C 180,E1 11468.587,E2 11468.587} C_VEL
LIN {X 0,Y 557.252,Z 988.687,A -85,B 0,C 180,E1 11473.914,E2 11473.914} C_VEL
LIN {X 0,Y 569.908,Z 914.196,A -85,B 0,C 180,E1 11477.687,E2 11477.687} C_VEL
LIN {X 0,Y 574.48,Z 866.359,A -85,B 0,C 180,E1 11479.313,E2 11479.313} C_VEL
LIN {X 0,Y 537.219,Z 802.443,A -85,B 0,C 180,E1 11485.764,E2 11485.764} C_VEL
LIN {X 0,Y 514.123,Z 767.06,A -85,B 0,C 180,E1 11490.463,E2 11490.463} C_VEL
LIN {X 0,Y 514.01,Z 767.06,A -85,B 0,C 180,E1 11500.184,E2 11500.184} C_VEL
LIN {X 0,Y 514.355,Z 767.06,A -85,B 0,C 180,E1 11508.971,E2 11508.971} C_VEL
LIN {X 0,Y 515.354,Z 767.06,A -85,B 0,C 180,E1 11519.179,E2 11519.179} C_VEL
LIN {X 0,Y 514.361,Z 767.06,A -85,B 0,C 180,E1 11529.357,E2 11529.357} C_VEL
LIN {X 0,Y 514.046,Z 767.06,A -85,B 0,C 180,E1 11538.074,E2 11538.074} C_VEL
LIN {X 0,Y 513.901,Z 767.06,A -85,B 0,C 180,E1 11547.253,E2 11547.253} C_VEL
LIN {X 0,Y 513.993,Z 768.912,A -85,B 0,C 180,E1 11556.877,E2 11556.877} C_VEL
LIN {X 0,Y 553.662,Z 828.826,A -85,B 0,C 180,E1 11564.211,E2 11564.211} C_VEL
LIN {X 0,Y 574.575,Z 871.294,A -85,B 0,C 180,E1 11568.161,E2 11568.161} C_VEL
LIN {X 0,Y 564.407,Z 943.735,A -85,B 0,C 180,E1 11571.012,E2 11571.012} C_VEL
LIN {X 0,Y 550.928,Z 1011.578,A -85,B 0,C 180,E1 11575.341,E2 11575.341} C_VEL
LIN {X 0,Y 536.466,Z 1074.388,A -85,B 0,C 180,E1 11581.449,E2 11581.449} C_VEL
LIN {X 0,Y 524.771,Z 1126.498,A -85,B 0,C 180,E1 11588.991,E2 11588.991} C_VEL
LIN {X 0,Y 518.162,Z 1163.05,A -85,B 0,C 180,E1 11596.841,E2 11596.841} C_VEL
LIN {X 0,Y 515.643,Z 1184.951,A -85,B 0,C 180,E1 11604.047,E2 11604.047} C_VEL
LIN {X 0,Y 514.907,Z 1196.55,A -85,B 0,C 180,E1 11610.803,E2 11610.803} C_VEL
LIN {X 0,Y 514.773,Z 1199.883,A -85,B 0,C 180,E1 11617.58,E2 11617.58} C_VEL
LIN {X 0,Y 515.338,Z 1193.649,A -85,B 0,C 180,E1 11625.323,E2 11625.323} C_VEL
LIN {X 0,Y 517.068,Z 1173.554,A -85,B 0,C 180,E1 11634.014,E2 11634.014} C_VEL
LIN {X 0,Y 522.006,Z 1140.658,A -85,B 0,C 180,E1 11642.242,E2 11642.242} C_VEL
LIN {X 0,Y 532.035,Z 1093.496,A -85,B 0,C 180,E1 11650.04,E2 11650.04} C_VEL
LIN {X 0,Y 545.995,Z 1033.505,A -85,B 0,C 180,E1 11656.709,E2 11656.709} C_VEL
LIN {X 0,Y 560.408,Z 965.803,A -85,B 0,C 180,E1 11661.704,E2 11661.704} C_VEL
LIN {X 0,Y 572.358,Z 891.801,A -85,B 0,C 180,E1 11665.179,E2 11665.179} C_VEL
LIN {X 0,Y 574.545,Z 866.944,A -85,B 0,C 180,E1 11666.081,E2 11666.081} C_VEL
LIN {X 0,Y 548.829,Z 817.368,A -85,B 0,C 180,E1 11671.418,E2 11671.418} C_VEL
LIN {X 0,Y 518.091,Z 773.926,A -85,B 0,C 180,E1 11678.508,E2 11678.508} C_VEL
LIN {X 0,Y 514.128,Z 767.06,A -85,B 0,C 180,E1 11680.141,E2 11680.141} C_VEL
LIN {X 0,Y 514.96,Z 767.06,A -85,B 0,C 180,E1 11688.939,E2 11688.939} C_VEL
LIN {X 0,Y 514.696,Z 767.06,A -85,B 0,C 180,E1 11699.133,E2 11699.133} C_VEL
LIN {X 0,Y 514.379,Z 767.06,A -85,B 0,C 180,E1 11707.604,E2 11707.604} C_VEL
LIN {X 0,Y 514.034,Z 767.06,A -85,B 0,C 180,E1 11716.55,E2 11716.55} C_VEL
LIN {X 0,Y 513.76,Z 767.06,A -85,B 0,C 180,E1 11726.478,E2 11726.478} C_VEL
LIN {X 0,Y 514.376,Z 770.094,A -85,B 0,C 180,E1 11727.282,E2 11727.282} C_VEL
LIN {X 0,Y 540.299,Z 804.999,A -85,B 0,C 180,E1 11733.606,E2 11733.606} C_VEL
LIN {X 0,Y 569.589,Z 854.329,A -85,B 0,C 180,E1 11739.457,E2 11739.457} C_VEL
LIN {X 0,Y 576.083,Z 871.881,A -85,B 0,C 180,E1 11740.937,E2 11740.937} C_VEL
LIN {X 0,Y 566.094,Z 941.67,A -85,B 0,C 180,E1 11743.493,E2 11743.493} C_VEL
LIN {X 0,Y 552.339,Z 1012.459,A -85,B 0,C 180,E1 11747.752,E2 11747.752} C_VEL
LIN {X 0,Y 538.14,Z 1076.996,A -85,B 0,C 180,E1 11753.709,E2 11753.709} C_VEL
LIN {X 0,Y 526.561,Z 1129.979,A -85,B 0,C 180,E1 11760.952,E2 11760.952} C_VEL
LIN {X 0,Y 521.897,Z 1151.337,A -85,B 0,C 180,E1 11764.863,E2 11764.863} C_VEL
LIN {X 0,Y 511.848,Z 1167.636,A -85,B 0,C 180,E1 11768.19,E2 11768.19} C_VEL
LIN {X 0,Y 507.968,Z 1193.93,A -85,B 0,C 180,E1 11776.452,E2 11776.452} C_VEL
LIN {X 0,Y 507.049,Z 1206.804,A -85,B 0,C 180,E1 11784.031,E2 11784.031} C_VEL
LIN {X 0,Y 506.713,Z 1209.828,A -85,B 0,C 180,E1 11790.9,E2 11790.9} C_VEL
LIN {X 0,Y 507.489,Z 1203.421,A -85,B 0,C 180,E1 11798.64,E2 11798.64} C_VEL
LIN {X 0,Y 509.252,Z 1183.963,A -85,B 0,C 180,E1 11807.174,E2 11807.174} C_VEL
LIN {X 0,Y 514.148,Z 1152.082,A -85,B 0,C 180,E1 11815.381,E2 11815.381} C_VEL
LIN {X 0,Y 524.27,Z 1106.115,A -85,B 0,C 180,E1 11823.167,E2 11823.167} C_VEL
LIN {X 0,Y 538.131,Z 1048.185,A -85,B 0,C 180,E1 11829.814,E2 11829.814} C_VEL
LIN {X 0,Y 552.843,Z 981.337,A -85,B 0,C 180,E1 11834.94,E2 11834.94} C_VEL
LIN {X 0,Y 565.242,Z 907.004,A -85,B 0,C 180,E1 11838.549,E2 11838.549} C_VEL
LIN {X 0,Y 568.782,Z 870.007,A -85,B 0,C 180,E1 11839.816,E2 11839.816} C_VEL
LIN {X 0,Y 531.828,Z 805.66,A -85,B 0,C 180,E1 11846.478,E2 11846.478} C_VEL
LIN {X 0,Y 506.138,Z 767.06,A -85,B 0,C 180,E1 11851.846,E2 11851.846} C_VEL
LIN {X 0,Y 506.038,Z 767.06,A -85,B 0,C 180,E1 11861.678,E2 11861.678} C_VEL
LIN {X 0,Y 506.585,Z 767.06,A -85,B 0,C 180,E1 11870.543,E2 11870.543} C_VEL
LIN {X 0,Y 506.742,Z 767.06,A -85,B 0,C 180,E1 11880.88,E2 11880.88} C_VEL
LIN {X 0,Y 506.328,Z 767.06,A -85,B 0,C 180,E1 11889.507,E2 11889.507} C_VEL
LIN {X 0,Y 505.946,Z 767.06,A -85,B 0,C 180,E1 11899.023,E2 11899.023} C_VEL
LIN {X 0,Y 505.853,Z 767.06,A -85,B 0,C 180,E1 11907.724,E2 11907.724} C_VEL
LIN {X 0,Y 505.928,Z 768.869,A -85,B 0,C 180,E1 11915.413,E2 11915.413} C_VEL
LIN {X 0,Y 543.748,Z 824.964,A -85,B 0,C 180,E1 11922.805,E2 11922.805} C_VEL
LIN {X 0,Y 568.833,Z 873.907,A -85,B 0,C 180,E1 11927.637,E2 11927.637} C_VEL
LIN {X 0,Y 558.33,Z 945.658,A -85,B 0,C 180,E1 11930.518,E2 11930.518} C_VEL
LIN {X 0,Y 544.458,Z 1013.041,A -85,B 0,C 180,E1 11934.875,E2 11934.875} C_VEL
LIN {X 0,Y 529.269,Z 1076.197,A -85,B 0,C 180,E1 11941.129,E2 11941.129} C_VEL
LIN {X 0,Y 517.269,Z 1127.172,A -85,B 0,C 180,E1 11948.672,E2 11948.672} C_VEL
LIN {X 0,Y 510.346,Z 1163.479,A -85,B 0,C 180,E1 11956.636,E2 11956.636} C_VEL
LIN {X 0,Y 507.695,Z 1185.188,A -85,B 0,C 180,E1 11963.953,E2 11963.953} C_VEL
LIN {X 0,Y 506.925,Z 1196.654,A -85,B 0,C 180,E1 11970.815,E2 11970.815} C_VEL
LIN {X 0,Y 506.77,Z 1199.862,A -85,B 0,C 180,E1 11977.7,E2 11977.7} C_VEL
LIN {X 0,Y 507.368,Z 1193.491,A -85,B 0,C 180,E1 11985.569,E2 11985.569} C_VEL
LIN {X 0,Y 509.152,Z 1173.925,A -85,B 0,C 180,E1 11994.159,E2 11994.159} C_VEL
LIN {X 0,Y 514.211,Z 1141.82,A -85,B 0,C 180,E1 12002.393,E2 12002.393} C_VEL
LIN {X 0,Y 524.639,Z 1095.197,A -85,B 0,C 180,E1 12010.312,E2 12010.312} C_VEL
LIN {X 0,Y 538.907,Z 1036.61,A -85,B 0,C 180,E1 12016.988,E2 12016.988} C_VEL
LIN {X 0,Y 553.942,Z 969.658,A -85,B 0,C 180,E1 12022.079,E2 12022.079} C_VEL
LIN {X 0,Y 566.683,Z 895.184,A -85,B 0,C 180,E1 12025.683,E2 12025.683} C_VEL
LIN {X 0,Y 568.904,Z 870.065,A -85,B 0,C 180,E1 12026.64,E2 12026.64} C_VEL
LIN {X 0,Y 543.542,Z 820.397,A -85,B 0,C 180,E1 12032.197,E2 12032.197} C_VEL
LIN {X 0,Y 514.512,Z 780.179,A -85,B 0,C 180,E1 12039.149,E2 12039.149} C_VEL
LIN {X 0,Y 506.262,Z 767.06,A -85,B 0,C 180,E1 12042.09,E2 12042.09} C_VEL
LIN {X 0,Y 506.718,Z 767.06,A -85,B 0,C 180,E1 12050.5,E2 12050.5} C_VEL
LIN {X 0,Y 506.719,Z 767.06,A -85,B 0,C 180,E1 12059.12,E2 12059.12} C_VEL
LIN {X 0,Y 506.365,Z 767.06,A -85,B 0,C 180,E1 12067.725,E2 12067.725} C_VEL
LIN {X 0,Y 506.041,Z 767.06,A -85,B 0,C 180,E1 12076.522,E2 12076.522} C_VEL
LIN {X 0,Y 505.907,Z 768.71,A -85,B 0,C 180,E1 12085.032,E2 12085.032} C_VEL
LIN {X 0,Y 533.246,Z 805.816,A -85,B 0,C 180,E1 12092.351,E2 12092.351} C_VEL
LIN {X 0,Y 561.108,Z 851.805,A -85,B 0,C 180,E1 12098.237,E2 12098.237} C_VEL
LIN {X 0,Y 570.638,Z 875.179,A -85,B 0,C 180,E1 12100.402,E2 12100.402} C_VEL
LIN {X 0,Y 559.934,Z 945.411,A -85,B 0,C 180,E1 12103.055,E2 12103.055} C_VEL
LIN {X 0,Y 545.471,Z 1015.998,A -85,B 0,C 180,E1 12107.442,E2 12107.442} C_VEL
LIN {X 0,Y 530.738,Z 1079.796,A -85,B 0,C 180,E1 12113.505,E2 12113.505} C_VEL
LIN {X 0,Y 518.653,Z 1132.592,A -85,B 0,C 180,E1 12120.946,E2 12120.946} C_VEL
LIN {X 0,Y 511.848,Z 1167.636,A -85,B 0,C 180,E1 12128.19,E2 12128.19} C_VEL
LIN {X 0,Y 501.478,Z 1181.443,A -85,B 0,C 180,E1 12131.698,E2 12131.698} C_VEL
LIN {X 0,Y 499.539,Z 1202.221,A -85,B 0,C 180,E1 12140.427,E2 12140.427} C_VEL
LIN {X 0,Y 499.28,Z 1209.421,A -85,B 0,C 180,E1 12147.43,E2 12147.43} C_VEL
LIN {X 0,Y 499.241,Z 1208.338,A -85,B 0,C 180,E1 12154.401,E2 12154.401} C_VEL
LIN {X 0,Y 499.609,Z 1197.087,A -85,B 0,C 180,E1 12162.318,E2 12162.318} C_VEL
LIN {X 0,Y 502.617,Z 1174.491,A -85,B 0,C 180,E1 12170.359,E2 12170.359} C_VEL
LIN {X 0,Y 509.976,Z 1137.094,A -85,B 0,C 180,E1 12178.705,E2 12178.705} C_VEL
LIN {X 0,Y 522.611,Z 1085.02,A -85,B 0,C 180,E1 12186.422,E2 12186.422} C_VEL
LIN {X 0,Y 538.043,Z 1022.07,A -85,B 0,C 180,E1 12192.669,E2 12192.669} C_VEL
LIN {X 0,Y 552.74,Z 952.284,A -85,B 0,C 180,E1 12197.157,E2 12197.157} C_VEL
LIN {X 0,Y 563.389,Z 882.211,A -85,B 0,C 180,E1 12199.926,E2 12199.926} C_VEL
LIN {X 0,Y 562.063,Z 871.245,A -85,B 0,C 180,E1 12200.538,E2 12200.538} C_VEL
LIN {X 0,Y 525.995,Z 808.651,A -85,B 0,C 180,E1 12207.292,E2 12207.292} C_VEL
LIN {X 0,Y 498.109,Z 767.06,A -85,B 0,C 180,E1 12213.333,E2 12213.333} C_VEL
LIN {X 0,Y 498.126,Z 767.06,A -85,B 0,C 180,E1 12223.786,E2 12223.786} C_VEL
LIN {X 0,Y 498.557,Z 767.06,A -85,B 0,C 180,E1 12232.153,E2 12232.153} C_VEL
LIN {X 0,Y 498.734,Z 767.06,A -85,B 0,C 180,E1 12240.894,E2 12240.894} C_VEL
LIN {X 0,Y 498.312,Z 767.06,A -85,B 0,C 180,E1 12249.662,E2 12249.662} C_VEL
LIN {X 0,Y 497.975,Z 767.06,A -85,B 0,C 180,E1 12258.678,E2 12258.678} C_VEL
LIN {X 0,Y 497.786,Z 767.06,A -85,B 0,C 180,E1 12268.213,E2 12268.213} C_VEL
LIN {X 0,Y 497.968,Z 769.09,A -85,B 0,C 180,E1 12273.867,E2 12273.867} C_VEL
LIN {X 0,Y 533.381,Z 820.464,A -85,B 0,C 180,E1 12281.24,E2 12281.24} C_VEL
LIN {X 0,Y 563.192,Z 875.969,A -85,B 0,C 180,E1 12287.088,E2 12287.088} C_VEL
LIN {X 0,Y 552.104,Z 948.376,A -85,B 0,C 180,E1 12290.059,E2 12290.059} C_VEL
LIN {X 0,Y 537.723,Z 1015.471,A -85,B 0,C 180,E1 12294.486,E2 12294.486} C_VEL
LIN {X 0,Y 522.292,Z 1077.168,A -85,B 0,C 180,E1 12300.706,E2 12300.706} C_VEL
LIN {X 0,Y 509.782,Z 1127.911,A -85,B 0,C 180,E1 12308.343,E2 12308.343} C_VEL
LIN {X 0,Y 502.281,Z 1165.506,A -85,B 0,C 180,E1 12316.862,E2 12316.862} C_VEL
LIN {X 0,Y 499.619,Z 1187.266,A -85,B 0,C 180,E1 12324.73,E2 12324.73} C_VEL
LIN {X 0,Y 499.123,Z 1198.364,A -85,B 0,C 180,E1 12332.571,E2 12332.571} C_VEL
LIN {X 0,Y 498.871,Z 1198.352,A -85,B 0,C 180,E1 12341.358,E2 12341.358} C_VEL
LIN {X 0,Y 499.474,Z 1187.213,A -85,B 0,C 180,E1 12349.209,E2 12349.209} C_VEL
LIN {X 0,Y 502.414,Z 1165.685,A -85,B 0,C 180,E1 12356.989,E2 12356.989} C_VEL
LIN {X 0,Y 510.103,Z 1127.561,A -85,B 0,C 180,E1 12365.618,E2 12365.618} C_VEL
LIN {X 0,Y 522.842,Z 1075.598,A -85,B 0,C 180,E1 12373.395,E2 12373.395} C_VEL
LIN {X 0,Y 538.651,Z 1012.308,A -85,B 0,C 180,E1 12379.703,E2 12379.703} C_VEL
LIN {X 0,Y 553.901,Z 942.497,A -85,B 0,C 180,E1 12384.241,E2 12384.241} C_VEL
LIN {X 0,Y 563.48,Z 873.663,A -85,B 0,C 180,E1 12387.171,E2 12387.171} C_VEL
LIN {X 0,Y 539.617,Z 825.983,A -85,B 0,C 180,E1 12392.698,E2 12392.698} C_VEL
LIN {X 0,Y 511.943,Z 787.046,A -85,B 0,C 180,E1 12399.547,E2 12399.547} C_VEL
LIN {X 0,Y 498.515,Z 767.06,A -85,B 0,C 180,E1 12404.082,E2 12404.082} C_VEL
LIN {X 0,Y 498.457,Z 767.06,A -85,B 0,C 180,E1 12412.106,E2 12412.106} C_VEL
LIN {X 0,Y 498.721,Z 767.06,A -85,B 0,C 180,E1 12419.106,E2 12419.106} C_VEL
LIN {X 0,Y 498.345,Z 767.06,A -85,B 0,C 180,E1 12427.85,E2 12427.85} C_VEL
LIN {X 0,Y 498.004,Z 767.06,A -85,B 0,C 180,E1 12436.797,E2 12436.797} C_VEL
LIN {X 0,Y 498.043,Z 768.935,A -85,B 0,C 180,E1 12442.701,E2 12442.701} C_VEL
LIN {X 0,Y 523.871,Z 802.786,A -85,B 0,C 180,E1 12450.422,E2 12450.422} C_VEL
LIN {X 0,Y 552.887,Z 849.544,A -85,B 0,C 180,E1 12456.98,E2 12456.98} C_VEL
LIN {X 0,Y 565.02,Z 879.606,A -85,B 0,C 180,E1 12459.899,E2 12459.899} C_VEL
LIN {X 0,Y 553.979,Z 948.317,A -85,B 0,C 180,E1 12462.566,E2 12462.566} C_VEL
LIN {X 0,Y 538.824,Z 1018.755,A -85,B 0,C 180,E1 12467.059,E2 12467.059} C_VEL
LIN {X 0,Y 523.262,Z 1082.784,A -85,B 0,C 180,E1 12473.313,E2 12473.313} C_VEL
LIN {X 0,Y 511.037,Z 1133.824,A -85,B 0,C 180,E1 12480.715,E2 12480.715} C_VEL
LIN {X 0,Y 502.87,Z 1173.315,A -85,B 0,C 180,E1 12489.3,E2 12489.3} C_VEL
LIN {X 0,Y 501.478,Z 1181.443,A -85,B 0,C 180,E1 12491.698,E2 12491.698} C_VEL
LIN {X 0,Y 492.489,Z 1192.596,A -85,B 0,C 180,E1 12495.463,E2 12495.463} C_VEL
LIN {X 0,Y 491.086,Z 1206.798,A -85,B 0,C 180,E1 12503.836,E2 12503.836} C_VEL
LIN {X 0,Y 490.727,Z 1209.828,A -85,B 0,C 180,E1 12510.929,E2 12510.929} C_VEL
LIN {X 0,Y 491.519,Z 1203.71,A -85,B 0,C 180,E1 12518.706,E2 12518.706} C_VEL
LIN {X 0,Y 493.396,Z 1184.606,A -85,B 0,C 180,E1 12527.521,E2 12527.521} C_VEL
LIN {X 0,Y 499.118,Z 1151.977,A -85,B 0,C 180,E1 12536.202,E2 12536.202} C_VEL
LIN {X 0,Y 510.22,Z 1105.965,A -85,B 0,C 180,E1 12544.196,E2 12544.196} C_VEL
LIN {X 0,Y 525.475,Z 1047.655,A -85,B 0,C 180,E1 12551.006,E2 12551.006} C_VEL
LIN {X 0,Y 541.243,Z 980.649,A -85,B 0,C 180,E1 12556.174,E2 12556.174} C_VEL
LIN {X 0,Y 554.571,Z 905.189,A -85,B 0,C 180,E1 12559.831,E2 12559.831} C_VEL
LIN {X 0,Y 557.327,Z 876.86,A -85,B 0,C 180,E1 12560.865,E2 12560.865} C_VEL
LIN {X 0,Y 521.684,Z 813.45,A -85,B 0,C 180,E1 12567.852,E2 12567.852} C_VEL
LIN {X 0,Y 490.066,Z 767.06,A -85,B 0,C 180,E1 12575.325,E2 12575.325} C_VEL
LIN {X 0,Y 490.132,Z 767.06,A -85,B 0,C 180,E1 12584.772,E2 12584.772} C_VEL
LIN {X 0,Y 490.384,Z 767.06,A -85,B 0,C 180,E1 12593.808,E2 12593.808} C_VEL
LIN {X 0,Y 490.727,Z 767.06,A -85,B 0,C 180,E1 12600.909,E2 12600.909} C_VEL
LIN {X 0,Y 490.281,Z 767.06,A -85,B 0,C 180,E1 12609.821,E2 12609.821} C_VEL
LIN {X 0,Y 489.955,Z 767.06,A -85,B 0,C 180,E1 12619.043,E2 12619.043} C_VEL
LIN {X 0,Y 489.764,Z 767.06,A -85,B 0,C 180,E1 12628.717,E2 12628.717} C_VEL
LIN {X 0,Y 489.901,Z 768.798,A -85,B 0,C 180,E1 12632.155,E2 12632.155} C_VEL
LIN {X 0,Y 525.026,Z 819.105,A -85,B 0,C 180,E1 12639.956,E2 12639.956} C_VEL
LIN {X 0,Y 557.407,Z 879.421,A -85,B 0,C 180,E1 12646.57,E2 12646.57} C_VEL
LIN {X 0,Y 545.373,Z 953.592,A -85,B 0,C 180,E1 12649.721,E2 12649.721} C_VEL
LIN {X 0,Y 530.189,Z 1021.046,A -85,B 0,C 180,E1 12654.357,E2 12654.357} C_VEL
LIN {X 0,Y 514.191,Z 1082.382,A -85,B 0,C 180,E1 12660.817,E2 12660.817} C_VEL
LIN {X 0,Y 501.387,Z 1132.02,A -85,B 0,C 180,E1 12668.661,E2 12668.661} C_VEL
LIN {X 0,Y 494.176,Z 1167.341,A -85,B 0,C 180,E1 12677.094,E2 12677.094} C_VEL
LIN {X 0,Y 491.644,Z 1187.503,A -85,B 0,C 180,E1 12684.644,E2 12684.644} C_VEL
LIN {X 0,Y 491.141,Z 1198.429,A -85,B 0,C 180,E1 12692.612,E2 12692.612} C_VEL
LIN {X 0,Y 490.862,Z 1198.274,A -85,B 0,C 180,E1 12701.546,E2 12701.546} C_VEL
LIN {X 0,Y 491.638,Z 1186.61,A -85,B 0,C 180,E1 12709.698,E2 12709.698} C_VEL
LIN {X 0,Y 495.435,Z 1162.128,A -85,B 0,C 180,E1 12718.29,E2 12718.29} C_VEL
LIN {X 0,Y 504.353,Z 1121.82,A -85,B 0,C 180,E1 12727.114,E2 12727.114} C_VEL
LIN {X 0,Y 517.778,Z 1069.554,A -85,B 0,C 180,E1 12734.67,E2 12734.67} C_VEL
LIN {X 0,Y 534.221,Z 1005.829,A -85,B 0,C 180,E1 12740.837,E2 12740.837} C_VEL
LIN {X 0,Y 549.894,Z 935.354,A -85,B 0,C 180,E1 12745.238,E2 12745.238} C_VEL
LIN {X 0,Y 558.139,Z 877.416,A -85,B 0,C 180,E1 12747.701,E2 12747.701} C_VEL
LIN {X 0,Y 535.425,Z 831.186,A -85,B 0,C 180,E1 12753.242,E2 12753.242} C_VEL
LIN {X 0,Y 506.573,Z 789.223,A -85,B 0,C 180,E1 12760.841,E2 12760.841} C_VEL
LIN {X 0,Y 490.896,Z 767.06,A -85,B 0,C 180,E1 12767.046,E2 12767.046} C_VEL
LIN {X 0,Y 491.174,Z 767.06,A -85,B 0,C 180,E1 12777.321,E2 12777.321} C_VEL
LIN {X 0,Y 490.648,Z 767.06,A -85,B 0,C 180,E1 12786.189,E2 12786.189} C_VEL
LIN {X 0,Y 490.128,Z 767.06,A -85,B 0,C 180,E1 12795.228,E2 12795.228} C_VEL
LIN {X 0,Y 490.163,Z 769.053,A -85,B 0,C 180,E1 12799.955,E2 12799.955} C_VEL
LIN {X 0,Y 509.454,Z 794.263,A -85,B 0,C 180,E1 12806.872,E2 12806.872} C_VEL
LIN {X 0,Y 536.544,Z 832.888,A -85,B 0,C 180,E1 12813.74,E2 12813.74} C_VEL
LIN {X 0,Y 559.992,Z 880.031,A -85,B 0,C 180,E1 12819.261,E2 12819.261} C_VEL
LIN {X 0,Y 548.315,Z 950.007,A -85,B 0,C 180,E1 12822.007,E2 12822.007} C_VEL
LIN {X 0,Y 532.177,Z 1021.542,A -85,B 0,C 180,E1 12826.664,E2 12826.664} C_VEL
LIN {X 0,Y 516.041,Z 1084.509,A -85,B 0,C 180,E1 12832.985,E2 12832.985} C_VEL
LIN {X 0,Y 503.23,Z 1135.587,A -85,B 0,C 180,E1 12840.588,E2 12840.588} C_VEL
LIN {X 0,Y 494.824,Z 1174.794,A -85,B 0,C 180,E1 12849.398,E2 12849.398} C_VEL
LIN {X 0,Y 492.489,Z 1192.596,A -85,B 0,C 180,E1 12855.463,E2 12855.463} C_VEL
LIN {X 0,Y 483.476,Z 1200.955,A -85,B 0,C 180,E1 12859.371,E2 12859.371} C_VEL
LIN {X 0,Y 483.265,Z 1209.415,A -85,B 0,C 180,E1 12867.345,E2 12867.345} C_VEL
LIN {X 0,Y 483.221,Z 1208.332,A -85,B 0,C 180,E1 12874.547,E2 12874.547} C_VEL
LIN {X 0,Y 483.719,Z 1197.081,A -85,B 0,C 180,E1 12882.729,E2 12882.729} C_VEL
LIN {X 0,Y 487.574,Z 1172.878,A -85,B 0,C 180,E1 12891.495,E2 12891.495} C_VEL
LIN {X 0,Y 496.539,Z 1133.11,A -85,B 0,C 180,E1 12900.328,E2 12900.328} C_VEL
LIN {X 0,Y 510.448,Z 1080.356,A -85,B 0,C 180,E1 12908.081,E2 12908.081} C_VEL
LIN {X 0,Y 526.699,Z 1017.99,A -85,B 0,C 180,E1 12914.179,E2 12914.179} C_VEL
LIN {X 0,Y 542.246,Z 947.859,A -85,B 0,C 180,E1 12918.604,E2 12918.604} C_VEL
LIN {X 0,Y 551.595,Z 880.337,A -85,B 0,C 180,E1 12921.39,E2 12921.39} C_VEL
LIN {X 0,Y 517.319,Z 818.445,A -85,B 0,C 180,E1 12928.415,E2 12928.415} C_VEL
LIN {X 0,Y 485.472,Z 773.623,A -85,B 0,C 180,E1 12935.796,E2 12935.796} C_VEL
LIN {X 0,Y 481.97,Z 767.06,A -85,B 0,C 180,E1 12936.858,E2 12936.858} C_VEL
LIN {X 0,Y 482.131,Z 767.06,A -85,B 0,C 180,E1 12946.375,E2 12946.375} C_VEL
LIN {X 0,Y 482.348,Z 767.06,A -85,B 0,C 180,E1 12955.514,E2 12955.514} C_VEL
LIN {X 0,Y 482.467,Z 767.06,A -85,B 0,C 180,E1 12962.727,E2 12962.727} C_VEL
LIN {X 0,Y 482.178,Z 767.06,A -85,B 0,C 180,E1 12971.824,E2 12971.824} C_VEL
LIN {X 0,Y 481.873,Z 767.06,A -85,B 0,C 180,E1 12981.621,E2 12981.621} C_VEL
LIN {X 0,Y 481.901,Z 768.947,A -85,B 0,C 180,E1 12990.315,E2 12990.315} C_VEL
LIN {X 0,Y 515.377,Z 815.977,A -85,B 0,C 180,E1 12998.328,E2 12998.328} C_VEL
LIN {X 0,Y 547.795,Z 874.117,A -85,B 0,C 180,E1 13005.165,E2 13005.165} C_VEL
LIN {X 0,Y 551.2,Z 886.302,A -85,B 0,C 180,E1 13006.147,E2 13006.147} C_VEL
LIN {X 0,Y 538.44,Z 960.161,A -85,B 0,C 180,E1 13009.458,E2 13009.458} C_VEL
LIN {X 0,Y 522.455,Z 1027.462,A -85,B 0,C 180,E1 13014.302,E2 13014.302} C_VEL
LIN {X 0,Y 506.321,Z 1086.68,A -85,B 0,C 180,E1 13020.811,E2 13020.811} C_VEL
LIN {X 0,Y 493.316,Z 1134.94,A -85,B 0,C 180,E1 13028.768,E2 13028.768} C_VEL
LIN {X 0,Y 486.083,Z 1169.172,A -85,B 0,C 180,E1 13037.334,E2 13037.334} C_VEL
LIN {X 0,Y 483.595,Z 1189.508,A -85,B 0,C 180,E1 13045.457,E2 13045.457} C_VEL
LIN {X 0,Y 483.156,Z 1199.494,A -85,B 0,C 180,E1 13054.458,E2 13054.458} C_VEL
LIN {X 0,Y 483.049,Z 1196.478,A -85,B 0,C 180,E1 13063.58,E2 13063.58} C_VEL
LIN {X 0,Y 485.145,Z 1179.558,A -85,B 0,C 180,E1 13072.965,E2 13072.965} C_VEL
LIN {X 0,Y 490.538,Z 1147.628,A -85,B 0,C 180,E1 13082.394,E2 13082.394} C_VEL
LIN {X 0,Y 501.999,Z 1102.301,A -85,B 0,C 180,E1 13090.868,E2 13090.868} C_VEL
LIN {X 0,Y 518.304,Z 1044.108,A -85,B 0,C 180,E1 13098.076,E2 13098.076} C_VEL
LIN {X 0,Y 535.255,Z 978.559,A -85,B 0,C 180,E1 13103.458,E2 13103.458} C_VEL
LIN {X 0,Y 550.106,Z 904.99,A -85,B 0,C 180,E1 13107.276,E2 13107.276} C_VEL
LIN {X 0,Y 552.778,Z 881.032,A -85,B 0,C 180,E1 13108.261,E2 13108.261} C_VEL
LIN {X 0,Y 530.92,Z 835.79,A -85,B 0,C 180,E1 13113.869,E2 13113.869} C_VEL
LIN {X 0,Y 503.843,Z 796.111,A -85,B 0,C 180,E1 13121.328,E2 13121.328} C_VEL
LIN {X 0,Y 486.699,Z 773.88,A -85,B 0,C 180,E1 13127.978,E2 13127.978} C_VEL
LIN {X 0,Y 482.582,Z 767.06,A -85,B 0,C 180,E1 13130.934,E2 13130.934} C_VEL
LIN {X 0,Y 482.724,Z 767.06,A -85,B 0,C 180,E1 13139.076,E2 13139.076} C_VEL
LIN {X 0,Y 482.352,Z 767.06,A -85,B 0,C 180,E1 13148.112,E2 13148.112} C_VEL
LIN {X 0,Y 482.231,Z 769.013,A -85,B 0,C 180,E1 13156.506,E2 13156.506} C_VEL
LIN {X 0,Y 495.036,Z 785.696,A -85,B 0,C 180,E1 13162.438,E2 13162.438} C_VEL
LIN {X 0,Y 518.658,Z 816.678,A -85,B 0,C 180,E1 13169.743,E2 13169.743} C_VEL
LIN {X 0,Y 544.854,Z 861.455,A -85,B 0,C 180,E1 13176.247,E2 13176.247} C_VEL
LIN {X 0,Y 554.197,Z 886.129,A -85,B 0,C 180,E1 13178.777,E2 13178.777} C_VEL
LIN {X 0,Y 541.97,Z 955.21,A -85,B 0,C 180,E1 13181.636,E2 13181.636} C_VEL
LIN {X 0,Y 525.514,Z 1024.311,A -85,B 0,C 180,E1 13186.273,E2 13186.273} C_VEL
LIN {X 0,Y 508.857,Z 1086.18,A -85,B 0,C 180,E1 13192.642,E2 13192.642} C_VEL
LIN {X 0,Y 495.571,Z 1136.858,A -85,B 0,C 180,E1 13200.374,E2 13200.374} C_VEL
LIN {X 0,Y 487.104,Z 1174.771,A -85,B 0,C 180,E1 13209.057,E2 13209.057} C_VEL
LIN {X 0,Y 483.684,Z 1197.271,A -85,B 0,C 180,E1 13217.361,E2 13217.361} C_VEL
LIN {X 0,Y 483.476,Z 1200.955,A -85,B 0,C 180,E1 13219.371,E2 13219.371} C_VEL
LIN {X 0,Y 475.158,Z 1206.632,A -85,B 0,C 180,E1 13223.458,E2 13223.458} C_VEL
LIN {X 0,Y 474.739,Z 1209.828,A -85,B 0,C 180,E1 13230.961,E2 13230.961} C_VEL
LIN {X 0,Y 475.534,Z 1203.573,A -85,B 0,C 180,E1 13239.1,E2 13239.1} C_VEL
LIN {X 0,Y 477.633,Z 1184.849,A -85,B 0,C 180,E1 13248.021,E2 13248.021} C_VEL
LIN {X 0,Y 484.187,Z 1151.787,A -85,B 0,C 180,E1 13257.075,E2 13257.075} C_VEL
LIN {X 0,Y 496.699,Z 1104.715,A -85,B 0,C 180,E1 13265.437,E2 13265.437} C_VEL
LIN {X 0,Y 513.098,Z 1046.528,A -85,B 0,C 180,E1 13272.294,E2 13272.294} C_VEL
LIN {X 0,Y 530.109,Z 978.86,A -85,B 0,C 180,E1 13277.513,E2 13277.513} C_VEL
LIN {X 0,Y 544.122,Z 903.448,A -85,B 0,C 180,E1 13281.153,E2 13281.153} C_VEL
LIN {X 0,Y 545.86,Z 883.922,A -85,B 0,C 180,E1 13281.925,E2 13281.925} C_VEL
LIN {X 0,Y 513.421,Z 824.163,A -85,B 0,C 180,E1 13288.891,E2 13288.891} C_VEL
LIN {X 0,Y 482.891,Z 780.685,A -85,B 0,C 180,E1 13296.169,E2 13296.169} C_VEL
LIN {X 0,Y 473.912,Z 767.06,A -85,B 0,C 180,E1 13298.919,E2 13298.919} C_VEL
LIN {X 0,Y 474.198,Z 767.06,A -85,B 0,C 180,E1 13308.023,E2 13308.023} C_VEL
LIN {X 0,Y 475.317,Z 767.06,A -85,B 0,C 180,E1 13319.11,E2 13319.11} C_VEL
LIN {X 0,Y 474.533,Z 767.06,A -85,B 0,C 180,E1 13328.295,E2 13328.295} C_VEL
LIN {X 0,Y 473.98,Z 767.06,A -85,B 0,C 180,E1 13337.726,E2 13337.726} C_VEL
LIN {X 0,Y 473.669,Z 767.304,A -85,B 0,C 180,E1 13348.155,E2 13348.155} C_VEL
LIN {X 0,Y 510.049,Z 819.146,A -85,B 0,C 180,E1 13357.522,E2 13357.522} C_VEL
LIN {X 0,Y 541.383,Z 876.221,A -85,B 0,C 180,E1 13364.453,E2 13364.453} C_VEL
LIN {X 0,Y 545.362,Z 889.721,A -85,B 0,C 180,E1 13365.622,E2 13365.622} C_VEL
LIN {X 0,Y 532.012,Z 963.703,A -85,B 0,C 180,E1 13369.033,E2 13369.033} C_VEL
LIN {X 0,Y 515.613,Z 1030.142,A -85,B 0,C 180,E1 13373.931,E2 13373.931} C_VEL
LIN {X 0,Y 498.872,Z 1089.179,A -85,B 0,C 180,E1 13380.582,E2 13380.582} C_VEL
LIN {X 0,Y 485.529,Z 1136.745,A -85,B 0,C 180,E1 13388.651,E2 13388.651} C_VEL
LIN {X 0,Y 478.245,Z 1169.638,A -85,B 0,C 180,E1 13397.123,E2 13397.123} C_VEL
LIN {X 0,Y 475.604,Z 1189.7,A -85,B 0,C 180,E1 13405.38,E2 13405.38} C_VEL
LIN {X 0,Y 475.137,Z 1199.549,A -85,B 0,C 180,E1 13414.534,E2 13414.534} C_VEL
LIN {X 0,Y 475.089,Z 1196.365,A -85,B 0,C 180,E1 13423.812,E2 13423.812} C_VEL
LIN {X 0,Y 477.176,Z 1180.301,A -85,B 0,C 180,E1 13432.923,E2 13432.923} C_VEL
LIN {X 0,Y 482.421,Z 1150.498,A -85,B 0,C 180,E1 13442.134,E2 13442.134} C_VEL
LIN {X 0,Y 493.837,Z 1106.792,A -85,B 0,C 180,E1 13450.698,E2 13450.698} C_VEL
LIN {X 0,Y 510.432,Z 1050.027,A -85,B 0,C 180,E1 13458.086,E2 13458.086} C_VEL
LIN {X 0,Y 528.139,Z 984.986,A -85,B 0,C 180,E1 13463.688,E2 13463.688} C_VEL
LIN {X 0,Y 543.998,Z 911.534,A -85,B 0,C 180,E1 13467.684,E2 13467.684} C_VEL
LIN {X 0,Y 547.355,Z 884.089,A -85,B 0,C 180,E1 13468.879,E2 13468.879} C_VEL
LIN {X 0,Y 525.819,Z 839.374,A -85,B 0,C 180,E1 13474.678,E2 13474.678} C_VEL
LIN {X 0,Y 501.258,Z 802.94,A -85,B 0,C 180,E1 13481.791,E2 13481.791} C_VEL
LIN {X 0,Y 484.855,Z 781.3,A -85,B 0,C 180,E1 13488.357,E2 13488.357} C_VEL
LIN {X 0,Y 478.466,Z 773.948,A -85,B 0,C 180,E1 13491.974,E2 13491.974} C_VEL
LIN {X 0,Y 474.763,Z 767.06,A -85,B 0,C 180,E1 13495.394,E2 13495.394} C_VEL
LIN {X 0,Y 474.839,Z 767.06,A -85,B 0,C 180,E1 13504.557,E2 13504.557} C_VEL
LIN {X 0,Y 474.635,Z 769.201,A -85,B 0,C 180,E1 13511.848,E2 13511.848} C_VEL
LIN {X 0,Y 481.688,Z 778.827,A -85,B 0,C 180,E1 13516.85,E2 13516.85} C_VEL
LIN {X 0,Y 492.725,Z 792.237,A -85,B 0,C 180,E1 13521.953,E2 13521.953} C_VEL
LIN {X 0,Y 516.518,Z 824.595,A -85,B 0,C 180,E1 13529.56,E2 13529.56} C_VEL
LIN {X 0,Y 541.219,Z 868.275,A -85,B 0,C 180,E1 13535.986,E2 13535.986} C_VEL
LIN {X 0,Y 548.915,Z 889.502,A -85,B 0,C 180,E1 13538.208,E2 13538.208} C_VEL
LIN {X 0,Y 535.868,Z 959.209,A -85,B 0,C 180,E1 13541.189,E2 13541.189} C_VEL
LIN {X 0,Y 518.468,Z 1028.562,A -85,B 0,C 180,E1 13545.997,E2 13545.997} C_VEL
LIN {X 0,Y 500.62,Z 1091.425,A -85,B 0,C 180,E1 13552.742,E2 13552.742} C_VEL
LIN {X 0,Y 486.709,Z 1142.257,A -85,B 0,C 180,E1 13560.944,E2 13560.944} C_VEL
LIN {X 0,Y 478.565,Z 1178.23,A -85,B 0,C 180,E1 13569.781,E2 13569.781} C_VEL
LIN {X 0,Y 475.53,Z 1199.078,A -85,B 0,C 180,E1 13578.076,E2 13578.076} C_VEL
LIN {X 0,Y 475.158,Z 1206.632,A -85,B 0,C 180,E1 13583.458,E2 13583.458} C_VEL
LIN {X 0,Y 467.118,Z 1209.502,A -85,B 0,C 180,E1 13587.65,E2 13587.65} C_VEL
LIN {X 0,Y 467.191,Z 1208.326,A -85,B 0,C 180,E1 13594.703,E2 13594.703} C_VEL
LIN {X 0,Y 467.822,Z 1197.424,A -85,B 0,C 180,E1 13602.991,E2 13602.991} C_VEL
LIN {X 0,Y 472.201,Z 1172.692,A -85,B 0,C 180,E1 13612.231,E2 13612.231} C_VEL
LIN {X 0,Y 482.473,Z 1131.673,A -85,B 0,C 180,E1 13621.554,E2 13621.554} C_VEL
LIN {X 0,Y 497.416,Z 1079.584,A -85,B 0,C 180,E1 13629.323,E2 13629.323} C_VEL
LIN {X 0,Y 514.94,Z 1016.715,A -85,B 0,C 180,E1 13635.514,E2 13635.514} C_VEL
LIN {X 0,Y 531.532,Z 945.797,A -85,B 0,C 180,E1 13639.982,E2 13639.982} C_VEL
LIN {X 0,Y 540.277,Z 887.623,A -85,B 0,C 180,E1 13642.451,E2 13642.451} C_VEL
LIN {X 0,Y 508.577,Z 828.253,A -85,B 0,C 180,E1 13649.592,E2 13649.592} C_VEL
LIN {X 0,Y 479.643,Z 786.93,A -85,B 0,C 180,E1 13656.739,E2 13656.739} C_VEL
LIN {X 0,Y 465.932,Z 767.06,A -85,B 0,C 180,E1 13661.361,E2 13661.361} C_VEL
LIN {X 0,Y 466.529,Z 767.06,A -85,B 0,C 180,E1 13671.611,E2 13671.611} C_VEL
LIN {X 0,Y 466.705,Z 767.06,A -85,B 0,C 180,E1 13680.956,E2 13680.956} C_VEL
LIN {X 0,Y 466.212,Z 767.06,A -85,B 0,C 180,E1 13690.334,E2 13690.334} C_VEL
LIN {X 0,Y 465.877,Z 767.06,A -85,B 0,C 180,E1 13700.018,E2 13700.018} C_VEL
LIN {X 0,Y 465.884,Z 768.653,A -85,B 0,C 180,E1 13705.974,E2 13705.974} C_VEL
LIN {X 0,Y 495.941,Z 809.414,A -85,B 0,C 180,E1 13714.612,E2 13714.612} C_VEL
LIN {X 0,Y 526.262,Z 860.524,A -85,B 0,C 180,E1 13721.658,E2 13721.658} C_VEL
LIN {X 0,Y 539.924,Z 891.218,A -85,B 0,C 180,E1 13725.024,E2 13725.024} C_VEL
LIN {X 0,Y 525.994,Z 965.442,A -85,B 0,C 180,E1 13728.493,E2 13728.493} C_VEL
LIN {X 0,Y 508.97,Z 1031.927,A -85,B 0,C 180,E1 13733.476,E2 13733.476} C_VEL
LIN {X 0,Y 491.761,Z 1090.398,A -85,B 0,C 180,E1 13740.176,E2 13740.176} C_VEL
LIN {X 0,Y 478.033,Z 1137.392,A -85,B 0,C 180,E1 13748.299,E2 13748.299} C_VEL
LIN {X 0,Y 470.402,Z 1170.114,A -85,B 0,C 180,E1 13756.904,E2 13756.904} C_VEL
LIN {X 0,Y 467.614,Z 1189.892,A -85,B 0,C 180,E1 13765.301,E2 13765.301} C_VEL
LIN {X 0,Y 467.112,Z 1199.586,A -85,B 0,C 180,E1 13774.612,E2 13774.612} C_VEL
LIN {X 0,Y 467.114,Z 1196.253,A -85,B 0,C 180,E1 13784.053,E2 13784.053} C_VEL
LIN {X 0,Y 469.279,Z 1179.012,A -85,B 0,C 180,E1 13793.788,E2 13793.788} C_VEL
LIN {X 0,Y 475.127,Z 1149.278,A -85,B 0,C 180,E1 13802.886,E2 13802.886} C_VEL
LIN {X 0,Y 487.563,Z 1104.604,A -85,B 0,C 180,E1 13811.621,E2 13811.621} C_VEL
LIN {X 0,Y 505.315,Z 1046.886,A -85,B 0,C 180,E1 13819.077,E2 13819.077} C_VEL
LIN {X 0,Y 523.954,Z 980.75,A -85,B 0,C 180,E1 13824.659,E2 13824.659} C_VEL
LIN {X 0,Y 539.909,Z 907.594,A -85,B 0,C 180,E1 13828.54,E2 13828.54} C_VEL
LIN {X 0,Y 542.126,Z 887.877,A -85,B 0,C 180,E1 13829.443,E2 13829.443} C_VEL
LIN {X 0,Y 521.506,Z 844.131,A -85,B 0,C 180,E1 13835.316,E2 13835.316} C_VEL
LIN {X 0,Y 498.235,Z 809.086,A -85,B 0,C 180,E1 13842.422,E2 13842.422} C_VEL
LIN {X 0,Y 482.748,Z 788.47,A -85,B 0,C 180,E1 13848.879,E2 13848.879} C_VEL
LIN {X 0,Y 476.406,Z 781.255,A -85,B 0,C 180,E1 13852.658,E2 13852.658} C_VEL
LIN {X 0,Y 471.559,Z 774.216,A -85,B 0,C 180,E1 13857.21,E2 13857.21} C_VEL
LIN {X 0,Y 472.039,Z 774.745,A -85,B 0,C 180,E1 13870.156,E2 13870.156} C_VEL
LIN {X 0,Y 480.421,Z 786.732,A -85,B 0,C 180,E1 13876.721,E2 13876.721} C_VEL
LIN {X 0,Y 492.398,Z 801.919,A -85,B 0,C 180,E1 13882.266,E2 13882.266} C_VEL
LIN {X 0,Y 514.997,Z 833.464,A -85,B 0,C 180,E1 13889.547,E2 13889.547} C_VEL
LIN {X 0,Y 537.911,Z 875.898,A -85,B 0,C 180,E1 13895.828,E2 13895.828} C_VEL
LIN {X 0,Y 543.579,Z 893.669,A -85,B 0,C 180,E1 13897.653,E2 13897.653} C_VEL
LIN {X 0,Y 529.824,Z 962.773,A -85,B 0,C 180,E1 13900.696,E2 13900.696} C_VEL
LIN {X 0,Y 512.078,Z 1030.542,A -85,B 0,C 180,E1 13905.511,E2 13905.511} C_VEL
LIN {X 0,Y 494.065,Z 1091.443,A -85,B 0,C 180,E1 13912.161,E2 13912.161} C_VEL
LIN {X 0,Y 479.527,Z 1141.861,A -85,B 0,C 180,E1 13920.404,E2 13920.404} C_VEL
LIN {X 0,Y 470.793,Z 1178.362,A -85,B 0,C 180,E1 13929.505,E2 13929.505} C_VEL
LIN {X 0,Y 467.589,Z 1199.075,A -85,B 0,C 180,E1 13937.871,E2 13937.871} C_VEL
LIN {X 0,Y 467.163,Z 1208.376,A -85,B 0,C 180,E1 13945.389,E2 13945.389} C_VEL
LIN {X 0,Y 467.118,Z 1209.502,A -85,B 0,C 180,E1 13947.65,E2 13947.65} C_VEL
LIN {X 0,Y 458.883,Z 1209.6,A -85,B 0,C 180,E1 13951.909,E2 13951.909} C_VEL
LIN {X 0,Y 459.638,Z 1202.001,A -85,B 0,C 180,E1 13960.508,E2 13960.508} C_VEL
LIN {X 0,Y 462.333,Z 1181.769,A -85,B 0,C 180,E1 13969.706,E2 13969.706} C_VEL
LIN {X 0,Y 470.466,Z 1147.324,A -85,B 0,C 180,E1 13978.956,E2 13978.956} C_VEL
LIN {X 0,Y 484.416,Z 1100.141,A -85,B 0,C 180,E1 13987.212,E2 13987.212} C_VEL
LIN {X 0,Y 502.3,Z 1040.813,A -85,B 0,C 180,E1 13994.067,E2 13994.067} C_VEL
LIN {X 0,Y 519.947,Z 974.014,A -85,B 0,C 180,E1 13999.09,E2 13999.09} C_VEL
LIN {X 0,Y 534.24,Z 900.457,A -85,B 0,C 180,E1 14002.552,E2 14002.552} C_VEL
LIN {X 0,Y 534.019,Z 889.909,A -85,B 0,C 180,E1 14003.151,E2 14003.151} C_VEL
LIN {X 0,Y 503.405,Z 831.715,A -85,B 0,C 180,E1 14010.397,E2 14010.397} C_VEL
LIN {X 0,Y 473.876,Z 788.97,A -85,B 0,C 180,E1 14018.117,E2 14018.117} C_VEL
LIN {X 0,Y 458.054,Z 767.06,A -85,B 0,C 180,E1 14024.205,E2 14024.205} C_VEL
LIN {X 0,Y 458.428,Z 767.06,A -85,B 0,C 180,E1 14033.374,E2 14033.374} C_VEL
LIN {X 0,Y 458.711,Z 767.06,A -85,B 0,C 180,E1 14040.972,E2 14040.972} C_VEL
LIN {X 0,Y 458.184,Z 767.06,A -85,B 0,C 180,E1 14050.517,E2 14050.517} C_VEL
LIN {X 0,Y 457.86,Z 767.06,A -85,B 0,C 180,E1 14060.384,E2 14060.384} C_VEL
LIN {X 0,Y 457.964,Z 768.816,A -85,B 0,C 180,E1 14063.384,E2 14063.384} C_VEL
LIN {X 0,Y 483.958,Z 803.111,A -85,B 0,C 180,E1 14071.896,E2 14071.896} C_VEL
LIN {X 0,Y 513.38,Z 849.665,A -85,B 0,C 180,E1 14079.196,E2 14079.196} C_VEL
LIN {X 0,Y 534.163,Z 894.631,A -85,B 0,C 180,E1 14084.476,E2 14084.476} C_VEL
LIN {X 0,Y 519.701,Z 968.544,A -85,B 0,C 180,E1 14088.029,E2 14088.029} C_VEL
LIN {X 0,Y 502.115,Z 1034.492,A -85,B 0,C 180,E1 14093.086,E2 14093.086} C_VEL
LIN {X 0,Y 484.223,Z 1093.026,A -85,B 0,C 180,E1 14099.972,E2 14099.972} C_VEL
LIN {X 0,Y 469.936,Z 1140.102,A -85,B 0,C 180,E1 14108.404,E2 14108.404} C_VEL
LIN {X 0,Y 462.337,Z 1172.019,A -85,B 0,C 180,E1 14117.154,E2 14117.154} C_VEL
LIN {X 0,Y 459.731,Z 1191.646,A -85,B 0,C 180,E1 14126.169,E2 14126.169} C_VEL
LIN {X 0,Y 459.109,Z 1199.608,A -85,B 0,C 180,E1 14134.692,E2 14134.692} C_VEL
LIN {X 0,Y 459.174,Z 1196.158,A -85,B 0,C 180,E1 14144.301,E2 14144.301} C_VEL
LIN {X 0,Y 461.296,Z 1179.975,A -85,B 0,C 180,E1 14153.706,E2 14153.706} C_VEL
LIN {X 0,Y 467.191,Z 1151.166,A -85,B 0,C 180,E1 14162.875,E2 14162.875} C_VEL
LIN {X 0,Y 480.202,Z 1106.395,A -85,B 0,C 180,E1 14171.922,E2 14171.922} C_VEL
LIN {X 0,Y 498.301,Z 1050.064,A -85,B 0,C 180,E1 14179.405,E2 14179.405} C_VEL
LIN {X 0,Y 517.719,Z 984.127,A -85,B 0,C 180,E1 14185.128,E2 14185.128} C_VEL
LIN {X 0,Y 534.48,Z 911.12,A -85,B 0,C 180,E1 14189.096,E2 14189.096} C_VEL
LIN {X 0,Y 537.188,Z 892.56,A -85,B 0,C 180,E1 14189.902,E2 14189.902} C_VEL
LIN {X 0,Y 516.92,Z 848.239,A -85,B 0,C 180,E1 14196.063,E2 14196.063} C_VEL
LIN {X 0,Y 492.892,Z 811.279,A -85,B 0,C 180,E1 14203.953,E2 14203.953} C_VEL
LIN {X 0,Y 477.597,Z 790.373,A -85,B 0,C 180,E1 14211.298,E2 14211.298} C_VEL
LIN {X 0,Y 469.992,Z 781.952,A -85,B 0,C 180,E1 14217.917,E2 14217.917} C_VEL
LIN {X 0,Y 471.767,Z 782.945,A -85,B 0,C 180,E1 14230.864,E2 14230.864} C_VEL
LIN {X 0,Y 484.603,Z 801.375,A -85,B 0,C 180,E1 14239.401,E2 14239.401} C_VEL
LIN {X 0,Y 504.939,Z 829.153,A -85,B 0,C 180,E1 14247.02,E2 14247.02} C_VEL
LIN {X 0,Y 528.136,Z 869.355,A -85,B 0,C 180,E1 14253.85,E2 14253.85} C_VEL
LIN {X 0,Y 538.293,Z 896.968,A -85,B 0,C 180,E1 14257.067,E2 14257.067} C_VEL
LIN {X 0,Y 524.02,Z 965.783,A -85,B 0,C 180,E1 14260.169,E2 14260.169} C_VEL
LIN {X 0,Y 505.246,Z 1034.308,A -85,B 0,C 180,E1 14265.173,E2 14265.173} C_VEL
LIN {X 0,Y 486.292,Z 1095.187,A -85,B 0,C 180,E1 14272.046,E2 14272.046} C_VEL
LIN {X 0,Y 471.161,Z 1145.418,A -85,B 0,C 180,E1 14280.64,E2 14280.64} C_VEL
LIN {X 0,Y 462.551,Z 1180.661,A -85,B 0,C 180,E1 14289.903,E2 14289.903} C_VEL
LIN {X 0,Y 459.52,Z 1200.57,A -85,B 0,C 180,E1 14298.621,E2 14298.621} C_VEL
LIN {X 0,Y 459.241,Z 1209.406,A -85,B 0,C 180,E1 14307.206,E2 14307.206} C_VEL
LIN {X 0,Y 458.883,Z 1209.6,A -85,B 0,C 180,E1 14311.909,E2 14311.909} C_VEL
LIN {X 0,Y 451.109,Z 1207.058,A -85,B 0,C 180,E1 14316.274,E2 14316.274} C_VEL
LIN {X 0,Y 452.903,Z 1192.928,A -85,B 0,C 180,E1 14325.595,E2 14325.595} C_VEL
LIN {X 0,Y 458.892,Z 1163.659,A -85,B 0,C 180,E1 14335.508,E2 14335.508} C_VEL
LIN {X 0,Y 471.5,Z 1120.014,A -85,B 0,C 180,E1 14344.685,E2 14344.685} C_VEL
LIN {X 0,Y 488.874,Z 1065.169,A -85,B 0,C 180,E1 14352.203,E2 14352.203} C_VEL
LIN {X 0,Y 507.27,Z 1001.327,A -85,B 0,C 180,E1 14357.977,E2 14357.977} C_VEL
LIN {X 0,Y 524.312,Z 927.389,A -85,B 0,C 180,E1 14362.176,E2 14362.176} C_VEL
LIN {X 0,Y 528.97,Z 894.788,A -85,B 0,C 180,E1 14363.572,E2 14363.572} C_VEL
LIN {X 0,Y 499.497,Z 837.396,A -85,B 0,C 180,E1 14370.892,E2 14370.892} C_VEL
LIN {X 0,Y 471.293,Z 795.951,A -85,B 0,C 180,E1 14378.549,E2 14378.549} C_VEL
LIN {X 0,Y 453.197,Z 773.44,A -85,B 0,C 180,E1 14385.268,E2 14385.268} C_VEL
LIN {X 0,Y 450.108,Z 767.06,A -85,B 0,C 180,E1 14387.372,E2 14387.372} C_VEL
LIN {X 0,Y 450.668,Z 767.06,A -85,B 0,C 180,E1 14397.131,E2 14397.131} C_VEL
LIN {X 0,Y 450.661,Z 767.06,A -85,B 0,C 180,E1 14406.791,E2 14406.791} C_VEL
LIN {X 0,Y 450.007,Z 767.06,A -85,B 0,C 180,E1 14416.677,E2 14416.677} C_VEL
LIN {X 0,Y 450.149,Z 769.189,A -85,B 0,C 180,E1 14420.365,E2 14420.365} C_VEL
LIN {X 0,Y 468.194,Z 792.742,A -85,B 0,C 180,E1 14427.59,E2 14427.59} C_VEL
LIN {X 0,Y 495.187,Z 831.013,A -85,B 0,C 180,E1 14435.212,E2 14435.212} C_VEL
LIN {X 0,Y 523.276,Z 884.294,A -85,B 0,C 180,E1 14442.406,E2 14442.406} C_VEL
LIN {X 0,Y 528.308,Z 899.124,A -85,B 0,C 180,E1 14443.961,E2 14443.961} C_VEL
LIN {X 0,Y 512.945,Z 973.469,A -85,B 0,C 180,E1 14447.66,E2 14447.66} C_VEL
LIN {X 0,Y 494.405,Z 1039.95,A -85,B 0,C 180,E1 14452.969,E2 14452.969} C_VEL
LIN {X 0,Y 475.977,Z 1098.121,A -85,B 0,C 180,E1 14460.139,E2 14460.139} C_VEL
LIN {X 0,Y 461.598,Z 1143.853,A -85,B 0,C 180,E1 14468.754,E2 14468.754} C_VEL
LIN {X 0,Y 454.014,Z 1175.028,A -85,B 0,C 180,E1 14477.896,E2 14477.896} C_VEL
LIN {X 0,Y 451.832,Z 1193.348,A -85,B 0,C 180,E1 14487.065,E2 14487.065} C_VEL
LIN {X 0,Y 451.083,Z 1199.699,A -85,B 0,C 180,E1 14494.776,E2 14494.776} C_VEL
LIN {X 0,Y 451.192,Z 1196.118,A -85,B 0,C 180,E1 14504.559,E2 14504.559} C_VEL
LIN {X 0,Y 453.438,Z 1179.598,A -85,B 0,C 180,E1 14514.205,E2 14514.205} C_VEL
LIN {X 0,Y 459.769,Z 1150.807,A -85,B 0,C 180,E1 14523.442,E2 14523.442} C_VEL
LIN {X 0,Y 473.291,Z 1106.817,A -85,B 0,C 180,E1 14532.469,E2 14532.469} C_VEL
LIN {X 0,Y 492.343,Z 1050.216,A -85,B 0,C 180,E1 14540.075,E2 14540.075} C_VEL
LIN {X 0,Y 512.056,Z 985.767,A -85,B 0,C 180,E1 14545.726,E2 14545.726} C_VEL
LIN {X 0,Y 529.624,Z 912.086,A -85,B 0,C 180,E1 14549.772,E2 14549.772} C_VEL
LIN {X 0,Y 531.994,Z 896.535,A -85,B 0,C 180,E1 14550.464,E2 14550.464} C_VEL
LIN {X 0,Y 513.163,Z 854.232,A -85,B 0,C 180,E1 14556.513,E2 14556.513} C_VEL
LIN {X 0,Y 490.606,Z 818.401,A -85,B 0,C 180,E1 14564.336,E2 14564.336} C_VEL
LIN {X 0,Y 475.868,Z 798,A -85,B 0,C 180,E1 14571.728,E2 14571.728} C_VEL
LIN {X 0,Y 469.013,Z 789.894,A -85,B 0,C 180,E1 14577.912,E2 14577.912} C_VEL
LIN {X 0,Y 470.595,Z 790.873,A -85,B 0,C 180,E1 14590.693,E2 14590.693} C_VEL
LIN {X 0,Y 483.509,Z 809.64,A -85,B 0,C 180,E1 14599.387,E2 14599.387} C_VEL
LIN {X 0,Y 504.186,Z 838.725,A -85,B 0,C 180,E1 14607.287,E2 14607.287} C_VEL
LIN {X 0,Y 526.393,Z 880.492,A -85,B 0,C 180,E1 14614.164,E2 14614.164} C_VEL
LIN {X 0,Y 533.209,Z 899.618,A -85,B 0,C 180,E1 14616.449,E2 14616.449} C_VEL
LIN {X 0,Y 518.507,Z 967.736,A -85,B 0,C 180,E1 14619.567,E2 14619.567} C_VEL
LIN {X 0,Y 499.079,Z 1035.828,A -85,B 0,C 180,E1 14624.62,E2 14624.62} C_VEL
LIN {X 0,Y 479.131,Z 1097.104,A -85,B 0,C 180,E1 14631.689,E2 14631.689} C_VEL
LIN {X 0,Y 463.561,Z 1146.328,A -85,B 0,C 180,E1 14640.356,E2 14640.356} C_VEL
LIN {X 0,Y 454.799,Z 1180.564,A -85,B 0,C 180,E1 14649.545,E2 14649.545} C_VEL
LIN {X 0,Y 451.56,Z 1200.479,A -85,B 0,C 180,E1 14658.418,E2 14658.418} C_VEL
LIN {X 0,Y 451.233,Z 1209.338,A -85,B 0,C 180,E1 14667.156,E2 14667.156} C_VEL
LIN {X 0,Y 451.109,Z 1207.058,A -85,B 0,C 180,E1 14676.274,E2 14676.274} C_VEL
LIN {X 0,Y 443.626,Z 1202.099,A -85,B 0,C 180,E1 14680.69,E2 14680.69} C_VEL
LIN {X 0,Y 446.501,Z 1182.938,A -85,B 0,C 180,E1 14689.917,E2 14689.917} C_VEL
LIN {X 0,Y 454.989,Z 1149.863,A -85,B 0,C 180,E1 14699.349,E2 14699.349} C_VEL
LIN {X 0,Y 470.103,Z 1102.606,A -85,B 0,C 180,E1 14708.012,E2 14708.012} C_VEL
LIN {X 0,Y 489.489,Z 1042.835,A -85,B 0,C 180,E1 14715.154,E2 14715.154} C_VEL
LIN {X 0,Y 508.336,Z 976.216,A -85,B 0,C 180,E1 14720.291,E2 14720.291} C_VEL
LIN {X 0,Y 523.765,Z 902.129,A -85,B 0,C 180,E1 14723.846,E2 14723.846} C_VEL
LIN {X 0,Y 500.066,Z 850.597,A -85,B 0,C 180,E1 14730.242,E2 14730.242} C_VEL
LIN {X 0,Y 472.675,Z 808.295,A -85,B 0,C 180,E1 14737.748,E2 14737.748} C_VEL
LIN {X 0,Y 451.915,Z 781.307,A -85,B 0,C 180,E1 14745.372,E2 14745.372} C_VEL
LIN {X 0,Y 442.455,Z 767.06,A -85,B 0,C 180,E1 14751.151,E2 14751.151} C_VEL
LIN {X 0,Y 442.72,Z 767.06,A -85,B 0,C 180,E1 14761.007,E2 14761.007} C_VEL
LIN {X 0,Y 442.144,Z 767.06,A -85,B 0,C 180,E1 14770.903,E2 14770.903} C_VEL
LIN {X 0,Y 442.293,Z 769.078,A -85,B 0,C 180,E1 14776.489,E2 14776.489} C_VEL
LIN {X 0,Y 454.849,Z 785.281,A -85,B 0,C 180,E1 14783.037,E2 14783.037} C_VEL
LIN {X 0,Y 478.729,Z 817.132,A -85,B 0,C 180,E1 14791.191,E2 14791.191} C_VEL
LIN {X 0,Y 505.829,Z 862.767,A -85,B 0,C 180,E1 14798.58,E2 14798.58} C_VEL
LIN {X 0,Y 522.791,Z 901.837,A -85,B 0,C 180,E1 14803.372,E2 14803.372} C_VEL
LIN {X 0,Y 506.719,Z 976.448,A -85,B 0,C 180,E1 14807.166,E2 14807.166} C_VEL
LIN {X 0,Y 487.545,Z 1042.668,A -85,B 0,C 180,E1 14812.582,E2 14812.582} C_VEL
LIN {X 0,Y 468.624,Z 1100.046,A -85,B 0,C 180,E1 14819.825,E2 14819.825} C_VEL
LIN {X 0,Y 453.815,Z 1145.515,A -85,B 0,C 180,E1 14828.628,E2 14828.628} C_VEL
LIN {X 0,Y 445.968,Z 1176.723,A -85,B 0,C 180,E1 14838.172,E2 14838.172} C_VEL
LIN {X 0,Y 443.754,Z 1194.757,A -85,B 0,C 180,E1 14847.992,E2 14847.992} C_VEL
LIN {X 0,Y 442.846,Z 1200.144,A -85,B 0,C 180,E1 14856.839,E2 14856.839} C_VEL
LIN {X 0,Y 443.322,Z 1194.902,A -85,B 0,C 180,E1 14865.81,E2 14865.81} C_VEL
LIN {X 0,Y 445.913,Z 1177.131,A -85,B 0,C 180,E1 14875.585,E2 14875.585} C_VEL
LIN {X 0,Y 453.502,Z 1147.029,A -85,B 0,C 180,E1 14884.92,E2 14884.92} C_VEL
LIN {X 0,Y 468.619,Z 1101.189,A -85,B 0,C 180,E1 14894.053,E2 14894.053} C_VEL
LIN {X 0,Y 489.054,Z 1042.626,A -85,B 0,C 180,E1 14901.6,E2 14901.6} C_VEL
LIN {X 0,Y 509.485,Z 977.289,A -85,B 0,C 180,E1 14907.024,E2 14907.024} C_VEL
LIN {X 0,Y 526.778,Z 903.553,A -85,B 0,C 180,E1 14910.848,E2 14910.848} C_VEL
